LIN {X 0,Y 389.933,Z 569.817,A -85,B 0,C 180,E1 -11709.597,E2 -11709.597} C_VEL
LIN {X 0,Y 390.463,Z 562.006,A -85,B 0,C 180,E1 -11711.157,E2 -11711.157} C_VEL
LIN {X 0,Y 391.267,Z 552.298,A -85,B 0,C 180,E1 -11712.711,E2 -11712.711} C_VEL
LIN {X 0,Y 392.166,Z 541.336,A -85,B 0,C 180,E1 -11714.133,E2 -11714.133} C_VEL
LIN {X 0,Y 392.924,Z 530.148,A -85,B 0,C 180,E1 -11715.299,E2 -11715.299} C_VEL
LIN {X 0,Y 393.801,Z 517.877,A -85,B 0,C 180,E1 -11716.325,E2 -11716.325} C_VEL
LIN {X 0,Y 394.289,Z 508.273,A -85,B 0,C 180,E1 -11716.971,E2 -11716.971} C_VEL
LIN {X 0,Y 391.847,Z 495.073,A -85,B 0,C 180,E1 -11717.783,E2 -11717.783} C_VEL
LIN {X 0,Y 389.258,Z 482.057,A -85,B 0,C 180,E1 -11718.418,E2 -11718.418} C_VEL
LIN {X 0,Y 389.378,Z 477.403,A -85,B 0,C 180,E1 -11721.161,E2 -11721.161} C_VEL
LIN {X 0,Y 389.588,Z 471.826,A -85,B 0,C 180,E1 -11724.514,E2 -11724.514} C_VEL
LIN {X 0,Y 389.891,Z 466.202,A -85,B 0,C 180,E1 -11727.961,E2 -11727.961} C_VEL
LIN {X 0,Y 390.122,Z 460.557,A -85,B 0,C 180,E1 -11731.496,E2 -11731.496} C_VEL
LIN {X 0,Y 390.336,Z 456.52,A -85,B 0,C 180,E1 -11734.081,E2 -11734.081} C_VEL
LIN {X 0,Y 390.324,Z 452.898,A -85,B 0,C 180,E1 -11736.455,E2 -11736.455} C_VEL
LIN {X 0,Y 390.174,Z 450.511,A -85,B 0,C 180,E1 -11738.092,E2 -11738.092} C_VEL
LIN {X 0,Y 390.038,Z 450.527,A -85,B 0,C 180,E1 -11741.813,E2 -11741.813} C_VEL
LIN {X 0,Y 390.052,Z 450.528,A -85,B 0,C 180,E1 -11745.354,E2 -11745.354} C_VEL
LIN {X 0,Y 390.08,Z 450.612,A -85,B 0,C 180,E1 -11748.317,E2 -11748.317} C_VEL
LIN {X 0,Y 391.012,Z 456.192,A -85,B 0,C 180,E1 -11751.016,E2 -11751.016} C_VEL
LIN {X 0,Y 391.083,Z 460.373,A -85,B 0,C 180,E1 -11752.984,E2 -11752.984} C_VEL
LIN {X 0,Y 390.807,Z 467.118,A -85,B 0,C 180,E1 -11756.117,E2 -11756.117} C_VEL
LIN {X 0,Y 390.549,Z 473.709,A -85,B 0,C 180,E1 -11759.144,E2 -11759.144} C_VEL
LIN {X 0,Y 390.319,Z 480.242,A -85,B 0,C 180,E1 -11762.084,E2 -11762.084} C_VEL
LIN {X 0,Y 390.081,Z 486.796,A -85,B 0,C 180,E1 -11764.95,E2 -11764.95} C_VEL
LIN {X 0,Y 389.917,Z 492.999,A -85,B 0,C 180,E1 -11767.561,E2 -11767.561} C_VEL
LIN {X 0,Y 394.076,Z 508.813,A -85,B 0,C 180,E1 -11768.244,E2 -11768.244} C_VEL
LIN {X 0,Y 396.749,Z 522.313,A -85,B 0,C 180,E1 -11768.978,E2 -11768.978} C_VEL
LIN {X 0,Y 397.539,Z 527.293,A -85,B 0,C 180,E1 -11769.293,E2 -11769.293} C_VEL
LIN {X 0,Y 396.695,Z 539.579,A -85,B 0,C 180,E1 -11770.041,E2 -11770.041} C_VEL
LIN {X 0,Y 395.73,Z 551.412,A -85,B 0,C 180,E1 -11770.953,E2 -11770.953} C_VEL
LIN {X 0,Y 394.45,Z 563.522,A -85,B 0,C 180,E1 -11772.099,E2 -11772.099} C_VEL
LIN {X 0,Y 393.359,Z 574.511,A -85,B 0,C 180,E1 -11773.388,E2 -11773.388} C_VEL
LIN {X 0,Y 392.11,Z 585.305,A -85,B 0,C 180,E1 -11774.935,E2 -11774.935} C_VEL
LIN {X 0,Y 391.204,Z 594.223,A -85,B 0,C 180,E1 -11776.493,E2 -11776.493} C_VEL
LIN {X 0,Y 390.405,Z 601.649,A -85,B 0,C 180,E1 -11778.051,E2 -11778.051} C_VEL
LIN {X 0,Y 389.812,Z 607.841,A -85,B 0,C 180,E1 -11779.612,E2 -11779.612} C_VEL
LIN {X 0,Y 389.208,Z 614.385,A -85,B 0,C 180,E1 -11781.693,E2 -11781.693} C_VEL
LIN {X 0,Y 388.924,Z 619.291,A -85,B 0,C 180,E1 -11783.774,E2 -11783.774} C_VEL
LIN {X 0,Y 388.707,Z 622.712,A -85,B 0,C 180,E1 -11785.851,E2 -11785.851} C_VEL
LIN {X 0,Y 388.654,Z 624.749,A -85,B 0,C 180,E1 -11787.926,E2 -11787.926} C_VEL
LIN {X 0,Y 388.672,Z 625.452,A -85,B 0,C 180,E1 -11789.999,E2 -11789.999} C_VEL
LIN {X 0,Y 388.653,Z 624.824,A -85,B 0,C 180,E1 -11792.071,E2 -11792.071} C_VEL
LIN {X 0,Y 388.705,Z 622.851,A -85,B 0,C 180,E1 -11794.146,E2 -11794.146} C_VEL
LIN {X 0,Y 388.902,Z 619.492,A -85,B 0,C 180,E1 -11796.223,E2 -11796.223} C_VEL
LIN {X 0,Y 389.189,Z 614.648,A -85,B 0,C 180,E1 -11798.305,E2 -11798.305} C_VEL
LIN {X 0,Y 389.754,Z 608.177,A -85,B 0,C 180,E1 -11800.387,E2 -11800.387} C_VEL
LIN {X 0,Y 390.448,Z 601.498,A -85,B 0,C 180,E1 -11802.08,E2 -11802.08} C_VEL
LIN {X 0,Y 390.181,Z 598.35,A -85,B 0,C 180,E1 -11802.813,E2 -11802.813} C_VEL
LIN {X 0,Y 387.895,Z 592.988,A -85,B 0,C 180,E1 -11803.997,E2 -11803.997} C_VEL
LIN {X 0,Y 385.67,Z 587.106,A -85,B 0,C 180,E1 -11805.136,E2 -11805.136} C_VEL
LIN {X 0,Y 385.494,Z 583.143,A -85,B 0,C 180,E1 -11805.787,E2 -11805.787} C_VEL
LIN {X 0,Y 386.652,Z 573.256,A -85,B 0,C 180,E1 -11807.178,E2 -11807.178} C_VEL
LIN {X 0,Y 387.927,Z 561.979,A -85,B 0,C 180,E1 -11808.483,E2 -11808.483} C_VEL
LIN {X 0,Y 389.194,Z 549.516,A -85,B 0,C 180,E1 -11809.652,E2 -11809.652} C_VEL
LIN {X 0,Y 390.291,Z 536.229,A -85,B 0,C 180,E1 -11810.642,E2 -11810.642} C_VEL
LIN {X 0,Y 390.728,Z 527.81,A -85,B 0,C 180,E1 -11811.156,E2 -11811.156} C_VEL
LIN {X 0,Y 388.377,Z 514.529,A -85,B 0,C 180,E1 -11811.963,E2 -11811.963} C_VEL
LIN {X 0,Y 384.932,Z 500.27,A -85,B 0,C 180,E1 -11812.667,E2 -11812.667} C_VEL
LIN {X 0,Y 382.917,Z 493.014,A -85,B 0,C 180,E1 -11812.972,E2 -11812.972} C_VEL
LIN {X 0,Y 383.224,Z 484.334,A -85,B 0,C 180,E1 -11816.698,E2 -11816.698} C_VEL
LIN {X 0,Y 383.47,Z 477.73,A -85,B 0,C 180,E1 -11819.657,E2 -11819.657} C_VEL
LIN {X 0,Y 383.735,Z 469.811,A -85,B 0,C 180,E1 -11823.327,E2 -11823.327} C_VEL
LIN {X 0,Y 384.019,Z 463.336,A -85,B 0,C 180,E1 -11826.365,E2 -11826.365} C_VEL
LIN {X 0,Y 384.18,Z 458.893,A -85,B 0,C 180,E1 -11828.459,E2 -11828.459} C_VEL
LIN {X 0,Y 383.663,Z 454.572,A -85,B 0,C 180,E1 -11830.55,E2 -11830.55} C_VEL
LIN {X 0,Y 383.079,Z 451.397,A -85,B 0,C 180,E1 -11832.214,E2 -11832.214} C_VEL
LIN {X 0,Y 383.066,Z 451.397,A -85,B 0,C 180,E1 -11835.799,E2 -11835.799} C_VEL
LIN {X 0,Y 383.037,Z 451.399,A -85,B 0,C 180,E1 -11838.785,E2 -11838.785} C_VEL
LIN {X 0,Y 382.995,Z 451.401,A -85,B 0,C 180,E1 -11842.094,E2 -11842.094} C_VEL
LIN {X 0,Y 383.01,Z 451.396,A -85,B 0,C 180,E1 -11845.331,E2 -11845.331} C_VEL
LIN {X 0,Y 383.028,Z 451.401,A -85,B 0,C 180,E1 -11847.852,E2 -11847.852} C_VEL
LIN {X 0,Y 383.055,Z 451.396,A -85,B 0,C 180,E1 -11851.719,E2 -11851.719} C_VEL
LIN {X 0,Y 383.043,Z 451.397,A -85,B 0,C 180,E1 -11855.039,E2 -11855.039} C_VEL
LIN {X 0,Y 383.012,Z 451.39,A -85,B 0,C 180,E1 -11858.47,E2 -11858.47} C_VEL
LIN {X 0,Y 383.084,Z 451.392,A -85,B 0,C 180,E1 -11861.827,E2 -11861.827} C_VEL
LIN {X 0,Y 383.104,Z 451.387,A -85,B 0,C 180,E1 -11865.118,E2 -11865.118} C_VEL
LIN {X 0,Y 383.098,Z 451.385,A -85,B 0,C 180,E1 -11868.358,E2 -11868.358} C_VEL
LIN {X 0,Y 383.293,Z 451.361,A -85,B 0,C 180,E1 -11871.932,E2 -11871.932} C_VEL
LIN {X 0,Y 383.197,Z 451.373,A -85,B 0,C 180,E1 -11874.738,E2 -11874.738} C_VEL
LIN {X 0,Y 383.378,Z 451.352,A -85,B 0,C 180,E1 -11877.899,E2 -11877.899} C_VEL
LIN {X 0,Y 383.51,Z 451.338,A -85,B 0,C 180,E1 -11880,E2 -11880} C_VEL
LIN {X 0,Y 383.243,Z 451.353,A -85,B 0,C 180,E1 -11883.154,E2 -11883.154} C_VEL
LIN {X 0,Y 383.277,Z 451.367,A -85,B 0,C 180,E1 -11886.316,E2 -11886.316} C_VEL
LIN {X 0,Y 383.25,Z 451.367,A -85,B 0,C 180,E1 -11888.436,E2 -11888.436} C_VEL
LIN {X 0,Y 383.098,Z 451.375,A -85,B 0,C 180,E1 -11891.642,E2 -11891.642} C_VEL
LIN {X 0,Y 383.101,Z 451.39,A -85,B 0,C 180,E1 -11894.882,E2 -11894.882} C_VEL
LIN {X 0,Y 383.052,Z 451.38,A -85,B 0,C 180,E1 -11898.174,E2 -11898.174} C_VEL
LIN {X 0,Y 382.986,Z 451.404,A -85,B 0,C 180,E1 -11901.531,E2 -11901.531} C_VEL
LIN {X 0,Y 383.042,Z 451.396,A -85,B 0,C 180,E1 -11904.961,E2 -11904.961} C_VEL
LIN {X 0,Y 383.04,Z 451.395,A -85,B 0,C 180,E1 -11908.493,E2 -11908.493} C_VEL
LIN {X 0,Y 382.997,Z 451.406,A -85,B 0,C 180,E1 -11912.428,E2 -11912.428} C_VEL
LIN {X 0,Y 383.018,Z 451.4,A -85,B 0,C 180,E1 -11915.956,E2 -11915.956} C_VEL
LIN {X 0,Y 383.014,Z 451.402,A -85,B 0,C 180,E1 -11919.589,E2 -11919.589} C_VEL
LIN {X 0,Y 383.057,Z 451.398,A -85,B 0,C 180,E1 -11922.789,E2 -11922.789} C_VEL
LIN {X 0,Y 383,Z 451.403,A -85,B 0,C 180,E1 -11925.792,E2 -11925.792} C_VEL
LIN {X 0,Y 383.053,Z 451.529,A -85,B 0,C 180,E1 -11928.664,E2 -11928.664} C_VEL
LIN {X 0,Y 384.348,Z 458.285,A -85,B 0,C 180,E1 -11931.839,E2 -11931.839} C_VEL
LIN {X 0,Y 385.925,Z 466.782,A -85,B 0,C 180,E1 -11935.632,E2 -11935.632} C_VEL
LIN {X 0,Y 386.157,Z 469.798,A -85,B 0,C 180,E1 -11936.909,E2 -11936.909} C_VEL
LIN {X 0,Y 385.52,Z 475.759,A -85,B 0,C 180,E1 -11939.309,E2 -11939.309} C_VEL
LIN {X 0,Y 384.58,Z 484.683,A -85,B 0,C 180,E1 -11942.817,E2 -11942.817} C_VEL
LIN {X 0,Y 383.72,Z 493.805,A -85,B 0,C 180,E1 -11946.316,E2 -11946.316} C_VEL
LIN {X 0,Y 383.49,Z 496.446,A -85,B 0,C 180,E1 -11947.314,E2 -11947.314} C_VEL
LIN {X 0,Y 387.196,Z 513.156,A -85,B 0,C 180,E1 -11947.964,E2 -11947.964} C_VEL
LIN {X 0,Y 389.483,Z 526.876,A -85,B 0,C 180,E1 -11948.659,E2 -11948.659} C_VEL
LIN {X 0,Y 390.207,Z 534.647,A -85,B 0,C 180,E1 -11949.116,E2 -11949.116} C_VEL
LIN {X 0,Y 389.251,Z 547.706,A -85,B 0,C 180,E1 -11949.939,E2 -11949.939} C_VEL
LIN {X 0,Y 388.105,Z 560.544,A -85,B 0,C 180,E1 -11950.978,E2 -11950.978} C_VEL
LIN {X 0,Y 386.84,Z 572.176,A -85,B 0,C 180,E1 -11952.148,E2 -11952.148} C_VEL
LIN {X 0,Y 385.572,Z 583.784,A -85,B 0,C 180,E1 -11953.591,E2 -11953.591} C_VEL
LIN {X 0,Y 384.448,Z 594.141,A -85,B 0,C 180,E1 -11955.173,E2 -11955.173} C_VEL
LIN {X 0,Y 383.595,Z 602.664,A -85,B 0,C 180,E1 -11956.762,E2 -11956.762} C_VEL
LIN {X 0,Y 382.78,Z 610.781,A -85,B 0,C 180,E1 -11958.618,E2 -11958.618} C_VEL
LIN {X 0,Y 382.232,Z 617.299,A -85,B 0,C 180,E1 -11960.476,E2 -11960.476} C_VEL
LIN {X 0,Y 381.842,Z 623.064,A -85,B 0,C 180,E1 -11962.599,E2 -11962.599} C_VEL
LIN {X 0,Y 381.754,Z 625.601,A -85,B 0,C 180,E1 -11963.787,E2 -11963.787} C_VEL
LIN {X 0,Y 381.628,Z 628.789,A -85,B 0,C 180,E1 -11965.777,E2 -11965.777} C_VEL
LIN {X 0,Y 381.574,Z 630.823,A -85,B 0,C 180,E1 -11967.89,E2 -11967.89} C_VEL
LIN {X 0,Y 381.604,Z 631.498,A -85,B 0,C 180,E1 -11970.001,E2 -11970.001} C_VEL
LIN {X 0,Y 381.579,Z 630.815,A -85,B 0,C 180,E1 -11972.112,E2 -11972.112} C_VEL
LIN {X 0,Y 381.629,Z 628.772,A -85,B 0,C 180,E1 -11974.226,E2 -11974.226} C_VEL
LIN {X 0,Y 381.765,Z 625.324,A -85,B 0,C 180,E1 -11976.343,E2 -11976.343} C_VEL
LIN {X 0,Y 381.977,Z 620.365,A -85,B 0,C 180,E1 -11978.466,E2 -11978.466} C_VEL
LIN {X 0,Y 382.355,Z 615.547,A -85,B 0,C 180,E1 -11980.058,E2 -11980.058} C_VEL
LIN {X 0,Y 383.057,Z 608.575,A -85,B 0,C 180,E1 -11981.913,E2 -11981.913} C_VEL
LIN {X 0,Y 383.826,Z 599.915,A -85,B 0,C 180,E1 -11983.772,E2 -11983.772} C_VEL
LIN {X 0,Y 384.846,Z 590.834,A -85,B 0,C 180,E1 -11985.356,E2 -11985.356} C_VEL
LIN {X 0,Y 386.088,Z 579.795,A -85,B 0,C 180,E1 -11986.934,E2 -11986.934} C_VEL
LIN {X 0,Y 387.284,Z 568.483,A -85,B 0,C 180,E1 -11988.243,E2 -11988.243} C_VEL
LIN {X 0,Y 388.505,Z 556.144,A -85,B 0,C 180,E1 -11989.397,E2 -11989.397} C_VEL
LIN {X 0,Y 390.036,Z 542.056,A -85,B 0,C 180,E1 -11990.572,E2 -11990.572} C_VEL
LIN {X 0,Y 390.784,Z 533.606,A -85,B 0,C 180,E1 -11991.161,E2 -11991.161} C_VEL
LIN {X 0,Y 389.733,Z 521.037,A -85,B 0,C 180,E1 -11992.054,E2 -11992.054} C_VEL
LIN {X 0,Y 387.574,Z 509.699,A -85,B 0,C 180,E1 -11992.827,E2 -11992.827} C_VEL
LIN {X 0,Y 384.121,Z 497.15,A -85,B 0,C 180,E1 -11993.666,E2 -11993.666} C_VEL
LIN {X 0,Y 385.4,Z 488.006,A -85,B 0,C 180,E1 -11997.712,E2 -11997.712} C_VEL
LIN {X 0,Y 386.913,Z 480.633,A -85,B 0,C 180,E1 -12001.381,E2 -12001.381} C_VEL
LIN {X 0,Y 387.785,Z 476.845,A -85,B 0,C 180,E1 -12003.521,E2 -12003.521} C_VEL
LIN {X 0,Y 387.574,Z 474.066,A -85,B 0,C 180,E1 -12005.47,E2 -12005.47} C_VEL
LIN {X 0,Y 387.084,Z 470.987,A -85,B 0,C 180,E1 -12008.121,E2 -12008.121} C_VEL
LIN {X 0,Y 386.649,Z 468.636,A -85,B 0,C 180,E1 -12010.873,E2 -12010.873} C_VEL
LIN {X 0,Y 386.265,Z 467.097,A -85,B 0,C 180,E1 -12013.742,E2 -12013.742} C_VEL
LIN {X 0,Y 386.086,Z 466.459,A -85,B 0,C 180,E1 -12016.731,E2 -12016.731} C_VEL
LIN {X 0,Y 386.06,Z 466.782,A -85,B 0,C 180,E1 -12019.872,E2 -12019.872} C_VEL
LIN {X 0,Y 386.068,Z 467.443,A -85,B 0,C 180,E1 -12021.761,E2 -12021.761} C_VEL
LIN {X 0,Y 385.8,Z 468.927,A -85,B 0,C 180,E1 -12024.343,E2 -12024.343} C_VEL
LIN {X 0,Y 385.177,Z 471.124,A -85,B 0,C 180,E1 -12027.07,E2 -12027.07} C_VEL
LIN {X 0,Y 384.481,Z 474.436,A -85,B 0,C 180,E1 -12030.427,E2 -12030.427} C_VEL
LIN {X 0,Y 383.857,Z 478.463,A -85,B 0,C 180,E1 -12033.934,E2 -12033.934} C_VEL
LIN {X 0,Y 383.328,Z 482.836,A -85,B 0,C 180,E1 -12037.355,E2 -12037.355} C_VEL
LIN {X 0,Y 383.139,Z 485.087,A -85,B 0,C 180,E1 -12039.017,E2 -12039.017} C_VEL
LIN {X 0,Y 384.261,Z 488.308,A -85,B 0,C 180,E1 -12039.289,E2 -12039.289} C_VEL
LIN {X 0,Y 388.12,Z 500.175,A -85,B 0,C 180,E1 -12040.325,E2 -12040.325} C_VEL
LIN {X 0,Y 390.526,Z 510.382,A -85,B 0,C 180,E1 -12041.23,E2 -12041.23} C_VEL
LIN {X 0,Y 390.913,Z 514.795,A -85,B 0,C 180,E1 -12041.608,E2 -12041.608} C_VEL
LIN {X 0,Y 389.458,Z 527.72,A -85,B 0,C 180,E1 -12042.677,E2 -12042.677} C_VEL
LIN {X 0,Y 388.138,Z 539.334,A -85,B 0,C 180,E1 -12043.877,E2 -12043.877} C_VEL
LIN {X 0,Y 386.703,Z 550.212,A -85,B 0,C 180,E1 -12045.26,E2 -12045.26} C_VEL
LIN {X 0,Y 385.608,Z 558.633,A -85,B 0,C 180,E1 -12046.563,E2 -12046.563} C_VEL
LIN {X 0,Y 384.546,Z 567.011,A -85,B 0,C 180,E1 -12048.135,E2 -12048.135} C_VEL
LIN {X 0,Y 383.756,Z 573.896,A -85,B 0,C 180,E1 -12049.714,E2 -12049.714} C_VEL
LIN {X 0,Y 382.955,Z 580.232,A -85,B 0,C 180,E1 -12051.558,E2 -12051.558} C_VEL
LIN {X 0,Y 382.505,Z 584.537,A -85,B 0,C 180,E1 -12053.185,E2 -12053.185} C_VEL
LIN {X 0,Y 382.048,Z 587.618,A -85,B 0,C 180,E1 -12054.723,E2 -12054.723} C_VEL
LIN {X 0,Y 382.067,Z 589.17,A -85,B 0,C 180,E1 -12055.781,E2 -12055.781} C_VEL
LIN {X 0,Y 381.973,Z 590.339,A -85,B 0,C 180,E1 -12056.836,E2 -12056.836} C_VEL
LIN {X 0,Y 381.821,Z 591.097,A -85,B 0,C 180,E1 -12057.89,E2 -12057.89} C_VEL
LIN {X 0,Y 381.728,Z 591.416,A -85,B 0,C 180,E1 -12058.945,E2 -12058.945} C_VEL
LIN {X 0,Y 381.696,Z 591.335,A -85,B 0,C 180,E1 -12060,E2 -12060} C_VEL
LIN {X 0,Y 381.709,Z 590.856,A -85,B 0,C 180,E1 -12061.055,E2 -12061.055} C_VEL
LIN {X 0,Y 381.788,Z 589.968,A -85,B 0,C 180,E1 -12062.11,E2 -12062.11} C_VEL
LIN {X 0,Y 381.806,Z 588.633,A -85,B 0,C 180,E1 -12063.166,E2 -12063.166} C_VEL
LIN {X 0,Y 381.888,Z 585.855,A -85,B 0,C 180,E1 -12064.75,E2 -12064.75} C_VEL
LIN {X 0,Y 382.163,Z 580.884,A -85,B 0,C 180,E1 -12066.745,E2 -12066.745} C_VEL
LIN {X 0,Y 382.469,Z 575.217,A -85,B 0,C 180,E1 -12068.453,E2 -12068.453} C_VEL
LIN {X 0,Y 382.975,Z 568.566,A -85,B 0,C 180,E1 -12070.04,E2 -12070.04} C_VEL
LIN {X 0,Y 383.561,Z 560.345,A -85,B 0,C 180,E1 -12071.628,E2 -12071.628} C_VEL
LIN {X 0,Y 384.471,Z 550.229,A -85,B 0,C 180,E1 -12073.209,E2 -12073.209} C_VEL
LIN {X 0,Y 385.38,Z 539.776,A -85,B 0,C 180,E1 -12074.522,E2 -12074.522} C_VEL
LIN {X 0,Y 386.158,Z 528.392,A -85,B 0,C 180,E1 -12075.694,E2 -12075.694} C_VEL
LIN {X 0,Y 386.979,Z 517.197,A -85,B 0,C 180,E1 -12076.621,E2 -12076.621} C_VEL
LIN {X 0,Y 387.398,Z 509.517,A -85,B 0,C 180,E1 -12077.145,E2 -12077.145} C_VEL
LIN {X 0,Y 385.102,Z 496.919,A -85,B 0,C 180,E1 -12077.959,E2 -12077.959} C_VEL
LIN {X 0,Y 382.409,Z 483.603,A -85,B 0,C 180,E1 -12078.622,E2 -12078.622} C_VEL
LIN {X 0,Y 382.182,Z 482.184,A -85,B 0,C 180,E1 -12078.703,E2 -12078.703} C_VEL
LIN {X 0,Y 382.336,Z 477.404,A -85,B 0,C 180,E1 -12081.57,E2 -12081.57} C_VEL
LIN {X 0,Y 382.498,Z 473.675,A -85,B 0,C 180,E1 -12083.843,E2 -12083.843} C_VEL
LIN {X 0,Y 382.761,Z 468.037,A -85,B 0,C 180,E1 -12087.325,E2 -12087.325} C_VEL
LIN {X 0,Y 383.028,Z 462.359,A -85,B 0,C 180,E1 -12090.915,E2 -12090.915} C_VEL
LIN {X 0,Y 383.226,Z 458.546,A -85,B 0,C 180,E1 -12093.379,E2 -12093.379} C_VEL
LIN {X 0,Y 383.3,Z 454.249,A -85,B 0,C 180,E1 -12096.218,E2 -12096.218} C_VEL
LIN {X 0,Y 383.137,Z 451.387,A -85,B 0,C 180,E1 -12098.213,E2 -12098.213} C_VEL
LIN {X 0,Y 382.991,Z 451.405,A -85,B 0,C 180,E1 -12101.347,E2 -12101.347} C_VEL
LIN {X 0,Y 383.004,Z 451.402,A -85,B 0,C 180,E1 -12104.303,E2 -12104.303} C_VEL
LIN {X 0,Y 383.057,Z 451.53,A -85,B 0,C 180,E1 -12108.045,E2 -12108.045} C_VEL
LIN {X 0,Y 384.027,Z 457.32,A -85,B 0,C 180,E1 -12110.9,E2 -12110.9} C_VEL
LIN {X 0,Y 384.114,Z 461.422,A -85,B 0,C 180,E1 -12112.857,E2 -12112.857} C_VEL
LIN {X 0,Y 383.819,Z 468.277,A -85,B 0,C 180,E1 -12116.078,E2 -12116.078} C_VEL
LIN {X 0,Y 383.514,Z 475.58,A -85,B 0,C 180,E1 -12119.462,E2 -12119.462} C_VEL
LIN {X 0,Y 383.243,Z 482.773,A -85,B 0,C 180,E1 -12122.711,E2 -12122.711} C_VEL
LIN {X 0,Y 382.989,Z 490.775,A -85,B 0,C 180,E1 -12126.189,E2 -12126.189} C_VEL
LIN {X 0,Y 382.919,Z 493.02,A -85,B 0,C 180,E1 -12127.135,E2 -12127.135} C_VEL
LIN {X 0,Y 386.942,Z 508.181,A -85,B 0,C 180,E1 -12127.8,E2 -12127.8} C_VEL
LIN {X 0,Y 389.679,Z 521.173,A -85,B 0,C 180,E1 -12128.521,E2 -12128.521} C_VEL
LIN {X 0,Y 390.802,Z 529.215,A -85,B 0,C 180,E1 -12129.028,E2 -12129.028} C_VEL
LIN {X 0,Y 389.839,Z 541.992,A -85,B 0,C 180,E1 -12129.854,E2 -12129.854} C_VEL
LIN {X 0,Y 388.754,Z 554.364,A -85,B 0,C 180,E1 -12130.871,E2 -12130.871} C_VEL
LIN {X 0,Y 387.376,Z 565.903,A -85,B 0,C 180,E1 -12132.035,E2 -12132.035} C_VEL
LIN {X 0,Y 386.297,Z 576.479,A -85,B 0,C 180,E1 -12133.348,E2 -12133.348} C_VEL
LIN {X 0,Y 385.065,Z 586.956,A -85,B 0,C 180,E1 -12134.924,E2 -12134.924} C_VEL
LIN {X 0,Y 384.253,Z 594.277,A -85,B 0,C 180,E1 -12136.244,E2 -12136.244} C_VEL
LIN {X 0,Y 383.449,Z 601.704,A -85,B 0,C 180,E1 -12137.831,E2 -12137.831} C_VEL
LIN {X 0,Y 382.791,Z 607.896,A -85,B 0,C 180,E1 -12139.419,E2 -12139.419} C_VEL
LIN {X 0,Y 382.154,Z 614.441,A -85,B 0,C 180,E1 -12141.538,E2 -12141.538} C_VEL
LIN {X 0,Y 381.85,Z 619.347,A -85,B 0,C 180,E1 -12143.659,E2 -12143.659} C_VEL
LIN {X 0,Y 381.636,Z 622.768,A -85,B 0,C 180,E1 -12145.774,E2 -12145.774} C_VEL
LIN {X 0,Y 381.552,Z 624.805,A -85,B 0,C 180,E1 -12147.887,E2 -12147.887} C_VEL
LIN {X 0,Y 381.572,Z 625.508,A -85,B 0,C 180,E1 -12149.999,E2 -12149.999} C_VEL
LIN {X 0,Y 381.551,Z 624.879,A -85,B 0,C 180,E1 -12152.11,E2 -12152.11} C_VEL
LIN {X 0,Y 381.634,Z 622.906,A -85,B 0,C 180,E1 -12154.223,E2 -12154.223} C_VEL
LIN {X 0,Y 381.848,Z 619.546,A -85,B 0,C 180,E1 -12156.339,E2 -12156.339} C_VEL
LIN {X 0,Y 382.137,Z 614.701,A -85,B 0,C 180,E1 -12158.459,E2 -12158.459} C_VEL
LIN {X 0,Y 382.74,Z 608.229,A -85,B 0,C 180,E1 -12160.579,E2 -12160.579} C_VEL
LIN {X 0,Y 383.564,Z 601.013,A -85,B 0,C 180,E1 -12162.431,E2 -12162.431} C_VEL
LIN {X 0,Y 384.351,Z 593.036,A -85,B 0,C 180,E1 -12164.101,E2 -12164.101} C_VEL
LIN {X 0,Y 385.494,Z 583.143,A -85,B 0,C 180,E1 -12165.787,E2 -12165.787} C_VEL
LIN {X 0,Y 385.351,Z 579.067,A -85,B 0,C 180,E1 -12166.424,E2 -12166.424} C_VEL
LIN {X 0,Y 383.287,Z 572.294,A -85,B 0,C 180,E1 -12167.463,E2 -12167.463} C_VEL
LIN {X 0,Y 381.343,Z 565.192,A -85,B 0,C 180,E1 -12168.45,E2 -12168.45} C_VEL
LIN {X 0,Y 381.35,Z 560.456,A -85,B 0,C 180,E1 -12168.986,E2 -12168.986} C_VEL
LIN {X 0,Y 382.663,Z 548.011,A -85,B 0,C 180,E1 -12170.141,E2 -12170.141} C_VEL
LIN {X 0,Y 383.686,Z 535.454,A -85,B 0,C 180,E1 -12171.072,E2 -12171.072} C_VEL
LIN {X 0,Y 384.069,Z 529.092,A -85,B 0,C 180,E1 -12171.466,E2 -12171.466} C_VEL
LIN {X 0,Y 381.721,Z 515.792,A -85,B 0,C 180,E1 -12172.313,E2 -12172.313} C_VEL
LIN {X 0,Y 378.38,Z 501.769,A -85,B 0,C 180,E1 -12173.041,E2 -12173.041} C_VEL
LIN {X 0,Y 375.878,Z 492.976,A -85,B 0,C 180,E1 -12173.446,E2 -12173.446} C_VEL
LIN {X 0,Y 376.208,Z 485.605,A -85,B 0,C 180,E1 -12176.636,E2 -12176.636} C_VEL
LIN {X 0,Y 376.479,Z 477.591,A -85,B 0,C 180,E1 -12180.265,E2 -12180.265} C_VEL
LIN {X 0,Y 376.86,Z 469.586,A -85,B 0,C 180,E1 -12184.017,E2 -12184.017} C_VEL
LIN {X 0,Y 377.192,Z 461.355,A -85,B 0,C 180,E1 -12187.94,E2 -12187.94} C_VEL
LIN {X 0,Y 377.139,Z 458.516,A -85,B 0,C 180,E1 -12189.313,E2 -12189.313} C_VEL
LIN {X 0,Y 376.037,Z 452.273,A -85,B 0,C 180,E1 -12192.459,E2 -12192.459} C_VEL
LIN {X 0,Y 375.994,Z 452.277,A -85,B 0,C 180,E1 -12196.243,E2 -12196.243} C_VEL
LIN {X 0,Y 375.992,Z 452.273,A -85,B 0,C 180,E1 -12200.026,E2 -12200.026} C_VEL
LIN {X 0,Y 375.957,Z 452.281,A -85,B 0,C 180,E1 -12203.494,E2 -12203.494} C_VEL
LIN {X 0,Y 375.952,Z 452.275,A -85,B 0,C 180,E1 -12205.888,E2 -12205.888} C_VEL
LIN {X 0,Y 375.966,Z 452.273,A -85,B 0,C 180,E1 -12209.687,E2 -12209.687} C_VEL
LIN {X 0,Y 375.993,Z 452.272,A -85,B 0,C 180,E1 -12212.141,E2 -12212.141} C_VEL
LIN {X 0,Y 375.997,Z 452.271,A -85,B 0,C 180,E1 -12214.538,E2 -12214.538} C_VEL
LIN {X 0,Y 375.975,Z 452.265,A -85,B 0,C 180,E1 -12218.046,E2 -12218.046} C_VEL
LIN {X 0,Y 376.022,Z 452.27,A -85,B 0,C 180,E1 -12221.474,E2 -12221.474} C_VEL
LIN {X 0,Y 376.052,Z 452.264,A -85,B 0,C 180,E1 -12224.832,E2 -12224.832} C_VEL
LIN {X 0,Y 376.049,Z 452.263,A -85,B 0,C 180,E1 -12228.136,E2 -12228.136} C_VEL
LIN {X 0,Y 376.247,Z 452.238,A -85,B 0,C 180,E1 -12231.876,E2 -12231.876} C_VEL
LIN {X 0,Y 376.169,Z 452.249,A -85,B 0,C 180,E1 -12234.64,E2 -12234.64} C_VEL
LIN {X 0,Y 376.344,Z 452.228,A -85,B 0,C 180,E1 -12237.859,E2 -12237.859} C_VEL
LIN {X 0,Y 376.48,Z 452.214,A -85,B 0,C 180,E1 -12240,E2 -12240} C_VEL
LIN {X 0,Y 376.181,Z 452.232,A -85,B 0,C 180,E1 -12243.213,E2 -12243.213} C_VEL
LIN {X 0,Y 376.236,Z 452.245,A -85,B 0,C 180,E1 -12246.435,E2 -12246.435} C_VEL
LIN {X 0,Y 376.195,Z 452.244,A -85,B 0,C 180,E1 -12248.595,E2 -12248.595} C_VEL
LIN {X 0,Y 376.05,Z 452.256,A -85,B 0,C 180,E1 -12251.863,E2 -12251.863} C_VEL
LIN {X 0,Y 376.049,Z 452.265,A -85,B 0,C 180,E1 -12255.168,E2 -12255.168} C_VEL
LIN {X 0,Y 375.998,Z 452.262,A -85,B 0,C 180,E1 -12258.527,E2 -12258.527} C_VEL
LIN {X 0,Y 375.954,Z 452.278,A -85,B 0,C 180,E1 -12261.955,E2 -12261.955} C_VEL
LIN {X 0,Y 375.996,Z 452.273,A -85,B 0,C 180,E1 -12265.462,E2 -12265.462} C_VEL
LIN {X 0,Y 375.967,Z 452.28,A -85,B 0,C 180,E1 -12269.079,E2 -12269.079} C_VEL
LIN {X 0,Y 375.945,Z 452.281,A -85,B 0,C 180,E1 -12272.829,E2 -12272.829} C_VEL
LIN {X 0,Y 375.949,Z 452.282,A -85,B 0,C 180,E1 -12275.416,E2 -12275.416} C_VEL
LIN {X 0,Y 375.969,Z 452.277,A -85,B 0,C 180,E1 -12278.272,E2 -12278.272} C_VEL
LIN {X 0,Y 375.982,Z 452.275,A -85,B 0,C 180,E1 -12281.611,E2 -12281.611} C_VEL
LIN {X 0,Y 375.961,Z 452.279,A -85,B 0,C 180,E1 -12285.263,E2 -12285.263} C_VEL
LIN {X 0,Y 376.006,Z 452.321,A -85,B 0,C 180,E1 -12288.292,E2 -12288.292} C_VEL
LIN {X 0,Y 377.269,Z 458.962,A -85,B 0,C 180,E1 -12291.481,E2 -12291.481} C_VEL
LIN {X 0,Y 378.663,Z 466.369,A -85,B 0,C 180,E1 -12294.877,E2 -12294.877} C_VEL
LIN {X 0,Y 379.179,Z 470.11,A -85,B 0,C 180,E1 -12296.519,E2 -12296.519} C_VEL
LIN {X 0,Y 378.477,Z 476.853,A -85,B 0,C 180,E1 -12299.295,E2 -12299.295} C_VEL
LIN {X 0,Y 377.519,Z 485.767,A -85,B 0,C 180,E1 -12302.867,E2 -12302.867} C_VEL
LIN {X 0,Y 376.537,Z 495.84,A -85,B 0,C 180,E1 -12306.805,E2 -12306.805} C_VEL
LIN {X 0,Y 376.516,Z 495.994,A -85,B 0,C 180,E1 -12306.864,E2 -12306.864} C_VEL
LIN {X 0,Y 380.27,Z 512.854,A -85,B 0,C 180,E1 -12307.53,E2 -12307.53} C_VEL
LIN {X 0,Y 382.547,Z 526.044,A -85,B 0,C 180,E1 -12308.214,E2 -12308.214} C_VEL
LIN {X 0,Y 383.481,Z 535.862,A -85,B 0,C 180,E1 -12308.809,E2 -12308.809} C_VEL
LIN {X 0,Y 382.426,Z 549.332,A -85,B 0,C 180,E1 -12309.697,E2 -12309.697} C_VEL
LIN {X 0,Y 381.211,Z 561.927,A -85,B 0,C 180,E1 -12310.761,E2 -12310.761} C_VEL
LIN {X 0,Y 379.945,Z 573.304,A -85,B 0,C 180,E1 -12311.953,E2 -12311.953} C_VEL
LIN {X 0,Y 378.723,Z 583.738,A -85,B 0,C 180,E1 -12313.285,E2 -12313.285} C_VEL
LIN {X 0,Y 377.544,Z 594.093,A -85,B 0,C 180,E1 -12314.895,E2 -12314.895} C_VEL
LIN {X 0,Y 376.613,Z 602.614,A -85,B 0,C 180,E1 -12316.512,E2 -12316.512} C_VEL
LIN {X 0,Y 375.963,Z 609.679,A -85,B 0,C 180,E1 -12318.135,E2 -12318.135} C_VEL
LIN {X 0,Y 375.328,Z 615.525,A -85,B 0,C 180,E1 -12319.755,E2 -12319.755} C_VEL
LIN {X 0,Y 374.824,Z 621.755,A -85,B 0,C 180,E1 -12321.917,E2 -12321.917} C_VEL
LIN {X 0,Y 374.681,Z 625.788,A -85,B 0,C 180,E1 -12323.792,E2 -12323.792} C_VEL
LIN {X 0,Y 374.554,Z 628.734,A -85,B 0,C 180,E1 -12325.697,E2 -12325.697} C_VEL
LIN {X 0,Y 374.471,Z 630.768,A -85,B 0,C 180,E1 -12327.85,E2 -12327.85} C_VEL
LIN {X 0,Y 374.505,Z 631.442,A -85,B 0,C 180,E1 -12330.001,E2 -12330.001} C_VEL
LIN {X 0,Y 374.476,Z 630.759,A -85,B 0,C 180,E1 -12332.152,E2 -12332.152} C_VEL
LIN {X 0,Y 374.555,Z 628.716,A -85,B 0,C 180,E1 -12334.306,E2 -12334.306} C_VEL
LIN {X 0,Y 374.678,Z 625.268,A -85,B 0,C 180,E1 -12336.463,E2 -12336.463} C_VEL
LIN {X 0,Y 374.937,Z 620.309,A -85,B 0,C 180,E1 -12338.626,E2 -12338.626} C_VEL
LIN {X 0,Y 375.325,Z 615.492,A -85,B 0,C 180,E1 -12340.248,E2 -12340.248} C_VEL
LIN {X 0,Y 376.071,Z 608.52,A -85,B 0,C 180,E1 -12342.138,E2 -12342.138} C_VEL
LIN {X 0,Y 376.878,Z 599.861,A -85,B 0,C 180,E1 -12344.031,E2 -12344.031} C_VEL
LIN {X 0,Y 377.949,Z 590.782,A -85,B 0,C 180,E1 -12345.643,E2 -12345.643} C_VEL
LIN {X 0,Y 379.272,Z 579.745,A -85,B 0,C 180,E1 -12347.248,E2 -12347.248} C_VEL
LIN {X 0,Y 380.541,Z 568.436,A -85,B 0,C 180,E1 -12348.578,E2 -12348.578} C_VEL
LIN {X 0,Y 382.625,Z 550.606,A -85,B 0,C 180,E1 -12350.32,E2 -12350.32} C_VEL
LIN {X 0,Y 384.035,Z 538.034,A -85,B 0,C 180,E1 -12351.33,E2 -12351.33} C_VEL
LIN {X 0,Y 384.284,Z 533.8,A -85,B 0,C 180,E1 -12351.637,E2 -12351.637} C_VEL
LIN {X 0,Y 383.237,Z 521.314,A -85,B 0,C 180,E1 -12352.571,E2 -12352.571} C_VEL
LIN {X 0,Y 380.871,Z 509.274,A -85,B 0,C 180,E1 -12353.447,E2 -12353.447} C_VEL
LIN {X 0,Y 377.305,Z 496.933,A -85,B 0,C 180,E1 -12354.347,E2 -12354.347} C_VEL
LIN {X 0,Y 378.649,Z 488.468,A -85,B 0,C 180,E1 -12358.25,E2 -12358.25} C_VEL
LIN {X 0,Y 380.166,Z 481.722,A -85,B 0,C 180,E1 -12361.746,E2 -12361.746} C_VEL
LIN {X 0,Y 380.903,Z 478.169,A -85,B 0,C 180,E1 -12363.871,E2 -12363.871} C_VEL
LIN {X 0,Y 380.583,Z 475.047,A -85,B 0,C 180,E1 -12366.224,E2 -12366.224} C_VEL
LIN {X 0,Y 380.106,Z 472.099,A -85,B 0,C 180,E1 -12369.053,E2 -12369.053} C_VEL
LIN {X 0,Y 379.744,Z 470.073,A -85,B 0,C 180,E1 -12371.78,E2 -12371.78} C_VEL
LIN {X 0,Y 379.35,Z 468.688,A -85,B 0,C 180,E1 -12375.251,E2 -12375.251} C_VEL
LIN {X 0,Y 379.235,Z 468.476,A -85,B 0,C 180,E1 -12378.152,E2 -12378.152} C_VEL
LIN {X 0,Y 379.218,Z 469.106,A -85,B 0,C 180,E1 -12381.114,E2 -12381.114} C_VEL
LIN {X 0,Y 379.043,Z 470.289,A -85,B 0,C 180,E1 -12383.607,E2 -12383.607} C_VEL
LIN {X 0,Y 378.492,Z 472.083,A -85,B 0,C 180,E1 -12386.148,E2 -12386.148} C_VEL
LIN {X 0,Y 377.911,Z 474.426,A -85,B 0,C 180,E1 -12388.812,E2 -12388.812} C_VEL
LIN {X 0,Y 377.174,Z 477.99,A -85,B 0,C 180,E1 -12392.236,E2 -12392.236} C_VEL
LIN {X 0,Y 376.555,Z 482.153,A -85,B 0,C 180,E1 -12395.757,E2 -12395.757} C_VEL
LIN {X 0,Y 376.216,Z 485.454,A -85,B 0,C 180,E1 -12398.313,E2 -12398.313} C_VEL
LIN {X 0,Y 377.397,Z 488.77,A -85,B 0,C 180,E1 -12398.612,E2 -12398.612} C_VEL
LIN {X 0,Y 381.522,Z 500.709,A -85,B 0,C 180,E1 -12399.742,E2 -12399.742} C_VEL
LIN {X 0,Y 384.021,Z 511.523,A -85,B 0,C 180,E1 -12400.767,E2 -12400.767} C_VEL
LIN {X 0,Y 384.529,Z 514.759,A -85,B 0,C 180,E1 -12401.076,E2 -12401.076} C_VEL
LIN {X 0,Y 383.223,Z 527.091,A -85,B 0,C 180,E1 -12402.111,E2 -12402.111} C_VEL
LIN {X 0,Y 381.645,Z 539.707,A -85,B 0,C 180,E1 -12403.432,E2 -12403.432} C_VEL
LIN {X 0,Y 380.287,Z 549.725,A -85,B 0,C 180,E1 -12404.731,E2 -12404.731} C_VEL
LIN {X 0,Y 378.804,Z 559.814,A -85,B 0,C 180,E1 -12406.317,E2 -12406.317} C_VEL
LIN {X 0,Y 377.697,Z 568.062,A -85,B 0,C 180,E1 -12407.917,E2 -12407.917} C_VEL
LIN {X 0,Y 376.829,Z 574.75,A -85,B 0,C 180,E1 -12409.523,E2 -12409.523} C_VEL
LIN {X 0,Y 375.99,Z 580.958,A -85,B 0,C 180,E1 -12411.4,E2 -12411.4} C_VEL
LIN {X 0,Y 375.572,Z 584.292,A -85,B 0,C 180,E1 -12412.654,E2 -12412.654} C_VEL
LIN {X 0,Y 375.003,Z 588.2,A -85,B 0,C 180,E1 -12414.623,E2 -12414.623} C_VEL
LIN {X 0,Y 375.005,Z 589.711,A -85,B 0,C 180,E1 -12415.701,E2 -12415.701} C_VEL
LIN {X 0,Y 374.921,Z 590.832,A -85,B 0,C 180,E1 -12416.776,E2 -12416.776} C_VEL
LIN {X 0,Y 374.762,Z 591.521,A -85,B 0,C 180,E1 -12417.851,E2 -12417.851} C_VEL
LIN {X 0,Y 374.627,Z 591.684,A -85,B 0,C 180,E1 -12420,E2 -12420} C_VEL
LIN {X 0,Y 374.643,Z 591.17,A -85,B 0,C 180,E1 -12421.075,E2 -12421.075} C_VEL
LIN {X 0,Y 374.707,Z 590.221,A -85,B 0,C 180,E1 -12422.15,E2 -12422.15} C_VEL
LIN {X 0,Y 374.711,Z 588.846,A -85,B 0,C 180,E1 -12423.226,E2 -12423.226} C_VEL
LIN {X 0,Y 374.829,Z 585.993,A -85,B 0,C 180,E1 -12424.84,E2 -12424.84} C_VEL
LIN {X 0,Y 375.092,Z 581.269,A -85,B 0,C 180,E1 -12426.753,E2 -12426.753} C_VEL
LIN {X 0,Y 375.41,Z 575.155,A -85,B 0,C 180,E1 -12428.614,E2 -12428.614} C_VEL
LIN {X 0,Y 375.952,Z 568.39,A -85,B 0,C 180,E1 -12430.23,E2 -12430.23} C_VEL
LIN {X 0,Y 376.576,Z 560.066,A -85,B 0,C 180,E1 -12431.847,E2 -12431.847} C_VEL
LIN {X 0,Y 377.35,Z 551.668,A -85,B 0,C 180,E1 -12433.188,E2 -12433.188} C_VEL
LIN {X 0,Y 378.239,Z 541.612,A -85,B 0,C 180,E1 -12434.52,E2 -12434.52} C_VEL
LIN {X 0,Y 379.071,Z 530.362,A -85,B 0,C 180,E1 -12435.732,E2 -12435.732} C_VEL
LIN {X 0,Y 379.987,Z 518.08,A -85,B 0,C 180,E1 -12436.798,E2 -12436.798} C_VEL
LIN {X 0,Y 380.432,Z 510.231,A -85,B 0,C 180,E1 -12437.354,E2 -12437.354} C_VEL
LIN {X 0,Y 377.992,Z 496.888,A -85,B 0,C 180,E1 -12438.232,E2 -12438.232} C_VEL
LIN {X 0,Y 375.246,Z 483.362,A -85,B 0,C 180,E1 -12438.913,E2 -12438.913} C_VEL
LIN {X 0,Y 375.119,Z 482.312,A -85,B 0,C 180,E1 -12438.998,E2 -12438.998} C_VEL
LIN {X 0,Y 375.313,Z 477.395,A -85,B 0,C 180,E1 -12441.994,E2 -12441.994} C_VEL
LIN {X 0,Y 375.542,Z 471.755,A -85,B 0,C 180,E1 -12445.495,E2 -12445.495} C_VEL
LIN {X 0,Y 375.846,Z 466.077,A -85,B 0,C 180,E1 -12449.09,E2 -12449.09} C_VEL
LIN {X 0,Y 376.153,Z 460.341,A -85,B 0,C 180,E1 -12452.809,E2 -12452.809} C_VEL
LIN {X 0,Y 376.248,Z 456.476,A -85,B 0,C 180,E1 -12455.384,E2 -12455.384} C_VEL
LIN {X 0,Y 376.104,Z 452.264,A -85,B 0,C 180,E1 -12458.294,E2 -12458.294} C_VEL
LIN {X 0,Y 375.938,Z 452.282,A -85,B 0,C 180,E1 -12462.3,E2 -12462.3} C_VEL
LIN {X 0,Y 375.96,Z 452.284,A -85,B 0,C 180,E1 -12465.264,E2 -12465.264} C_VEL
LIN {X 0,Y 376.024,Z 452.352,A -85,B 0,C 180,E1 -12467.711,E2 -12467.711} C_VEL
LIN {X 0,Y 377.02,Z 458.232,A -85,B 0,C 180,E1 -12470.668,E2 -12470.668} C_VEL
LIN {X 0,Y 377.154,Z 462.473,A -85,B 0,C 180,E1 -12472.722,E2 -12472.722} C_VEL
LIN {X 0,Y 376.846,Z 469.325,A -85,B 0,C 180,E1 -12475.978,E2 -12475.978} C_VEL
LIN {X 0,Y 376.482,Z 477.349,A -85,B 0,C 180,E1 -12479.732,E2 -12479.732} C_VEL
LIN {X 0,Y 376.186,Z 485.357,A -85,B 0,C 180,E1 -12483.359,E2 -12483.359} C_VEL
LIN {X 0,Y 375.929,Z 493.024,A -85,B 0,C 180,E1 -12486.685,E2 -12486.685} C_VEL
LIN {X 0,Y 380.041,Z 508.281,A -85,B 0,C 180,E1 -12487.378,E2 -12487.378} C_VEL
LIN {X 0,Y 382.773,Z 520.99,A -85,B 0,C 180,E1 -12488.103,E2 -12488.103} C_VEL
LIN {X 0,Y 384.074,Z 529.372,A -85,B 0,C 180,E1 -12488.651,E2 -12488.651} C_VEL
LIN {X 0,Y 383.147,Z 542.418,A -85,B 0,C 180,E1 -12489.518,E2 -12489.518} C_VEL
LIN {X 0,Y 382.037,Z 554.41,A -85,B 0,C 180,E1 -12490.522,E2 -12490.522} C_VEL
LIN {X 0,Y 380.495,Z 567.1,A -85,B 0,C 180,E1 -12491.837,E2 -12491.837} C_VEL
LIN {X 0,Y 379.234,Z 578.444,A -85,B 0,C 180,E1 -12493.306,E2 -12493.306} C_VEL
LIN {X 0,Y 377.995,Z 588.604,A -85,B 0,C 180,E1 -12494.911,E2 -12494.911} C_VEL
LIN {X 0,Y 377.215,Z 595.663,A -85,B 0,C 180,E1 -12496.257,E2 -12496.257} C_VEL
LIN {X 0,Y 376.326,Z 602.858,A -85,B 0,C 180,E1 -12497.871,E2 -12497.871} C_VEL
LIN {X 0,Y 375.586,Z 609.735,A -85,B 0,C 180,E1 -12499.759,E2 -12499.759} C_VEL
LIN {X 0,Y 375,Z 615.9,A -85,B 0,C 180,E1 -12501.918,E2 -12501.918} C_VEL
LIN {X 0,Y 374.768,Z 619.665,A -85,B 0,C 180,E1 -12503.673,E2 -12503.673} C_VEL
LIN {X 0,Y 374.566,Z 622.824,A -85,B 0,C 180,E1 -12505.694,E2 -12505.694} C_VEL
LIN {X 0,Y 374.45,Z 624.861,A -85,B 0,C 180,E1 -12507.847,E2 -12507.847} C_VEL
LIN {X 0,Y 374.473,Z 625.564,A -85,B 0,C 180,E1 -12509.999,E2 -12509.999} C_VEL
LIN {X 0,Y 374.449,Z 624.935,A -85,B 0,C 180,E1 -12512.15,E2 -12512.15} C_VEL
LIN {X 0,Y 374.564,Z 622.961,A -85,B 0,C 180,E1 -12514.303,E2 -12514.303} C_VEL
LIN {X 0,Y 374.78,Z 619.6,A -85,B 0,C 180,E1 -12516.459,E2 -12516.459} C_VEL
LIN {X 0,Y 375.098,Z 614.755,A -85,B 0,C 180,E1 -12518.619,E2 -12518.619} C_VEL
LIN {X 0,Y 375.709,Z 608.281,A -85,B 0,C 180,E1 -12520.78,E2 -12520.78} C_VEL
LIN {X 0,Y 376.598,Z 601.064,A -85,B 0,C 180,E1 -12522.665,E2 -12522.665} C_VEL
LIN {X 0,Y 377.539,Z 592.175,A -85,B 0,C 180,E1 -12524.534,E2 -12524.534} C_VEL
LIN {X 0,Y 378.703,Z 582.669,A -85,B 0,C 180,E1 -12526.161,E2 -12526.161} C_VEL
LIN {X 0,Y 379.986,Z 572.252,A -85,B 0,C 180,E1 -12527.628,E2 -12527.628} C_VEL
LIN {X 0,Y 381.35,Z 560.456,A -85,B 0,C 180,E1 -12528.986,E2 -12528.986} C_VEL
LIN {X 0,Y 381.348,Z 555.635,A -85,B 0,C 180,E1 -12529.502,E2 -12529.502} C_VEL
LIN {X 0,Y 379.375,Z 547.759,A -85,B 0,C 180,E1 -12530.369,E2 -12530.369} C_VEL
LIN {X 0,Y 377.324,Z 539.552,A -85,B 0,C 180,E1 -12531.158,E2 -12531.158} C_VEL
LIN {X 0,Y 377.181,Z 534.217,A -85,B 0,C 180,E1 -12531.541,E2 -12531.541} C_VEL
LIN {X 0,Y 377.231,Z 529.11,A -85,B 0,C 180,E1 -12531.875,E2 -12531.875} C_VEL
LIN {X 0,Y 374.758,Z 515.304,A -85,B 0,C 180,E1 -12532.772,E2 -12532.772} C_VEL
LIN {X 0,Y 371.308,Z 501.37,A -85,B 0,C 180,E1 -12533.515,E2 -12533.515} C_VEL
LIN {X 0,Y 368.906,Z 493.005,A -85,B 0,C 180,E1 -12533.903,E2 -12533.903} C_VEL
LIN {X 0,Y 369.229,Z 485.54,A -85,B 0,C 180,E1 -12537.18,E2 -12537.18} C_VEL
LIN {X 0,Y 369.481,Z 478.795,A -85,B 0,C 180,E1 -12540.267,E2 -12540.267} C_VEL
LIN {X 0,Y 369.882,Z 470.694,A -85,B 0,C 180,E1 -12544.09,E2 -12544.09} C_VEL
LIN {X 0,Y 370.18,Z 463.87,A -85,B 0,C 180,E1 -12547.409,E2 -12547.409} C_VEL
LIN {X 0,Y 370.134,Z 459.588,A -85,B 0,C 180,E1 -12549.498,E2 -12549.498} C_VEL
LIN {X 0,Y 368.997,Z 453.15,A -85,B 0,C 180,E1 -12552.792,E2 -12552.792} C_VEL
LIN {X 0,Y 368.968,Z 453.152,A -85,B 0,C 180,E1 -12556.368,E2 -12556.368} C_VEL
LIN {X 0,Y 368.945,Z 453.154,A -85,B 0,C 180,E1 -12559.634,E2 -12559.634} C_VEL
LIN {X 0,Y 368.895,Z 453.158,A -85,B 0,C 180,E1 -12563.143,E2 -12563.143} C_VEL
LIN {X 0,Y 368.891,Z 453.159,A -85,B 0,C 180,E1 -12566.461,E2 -12566.461} C_VEL
LIN {X 0,Y 368.919,Z 453.158,A -85,B 0,C 180,E1 -12570.31,E2 -12570.31} C_VEL
LIN {X 0,Y 368.972,Z 453.142,A -85,B 0,C 180,E1 -12573.534,E2 -12573.534} C_VEL
LIN {X 0,Y 368.969,Z 453.15,A -85,B 0,C 180,E1 -12576.422,E2 -12576.422} C_VEL
LIN {X 0,Y 368.946,Z 453.15,A -85,B 0,C 180,E1 -12579.947,E2 -12579.947} C_VEL
LIN {X 0,Y 368.969,Z 453.149,A -85,B 0,C 180,E1 -12583.398,E2 -12583.398} C_VEL
LIN {X 0,Y 369.049,Z 453.14,A -85,B 0,C 180,E1 -12586.79,E2 -12586.79} C_VEL
LIN {X 0,Y 369.062,Z 453.138,A -85,B 0,C 180,E1 -12590.131,E2 -12590.131} C_VEL
LIN {X 0,Y 369.178,Z 453.122,A -85,B 0,C 180,E1 -12592.342,E2 -12592.342} C_VEL
LIN {X 0,Y 369.142,Z 453.125,A -85,B 0,C 180,E1 -12594.537,E2 -12594.537} C_VEL
LIN {X 0,Y 369.309,Z 453.105,A -85,B 0,C 180,E1 -12597.819,E2 -12597.819} C_VEL
LIN {X 0,Y 369.449,Z 453.09,A -85,B 0,C 180,E1 -12600,E2 -12600} C_VEL
LIN {X 0,Y 369.309,Z 453.1,A -85,B 0,C 180,E1 -12602.181,E2 -12602.181} C_VEL
LIN {X 0,Y 369.198,Z 453.123,A -85,B 0,C 180,E1 -12606.558,E2 -12606.558} C_VEL
LIN {X 0,Y 369.128,Z 453.124,A -85,B 0,C 180,E1 -12608.761,E2 -12608.761} C_VEL
LIN {X 0,Y 369.004,Z 453.137,A -85,B 0,C 180,E1 -12612.093,E2 -12612.093} C_VEL
LIN {X 0,Y 368.988,Z 453.142,A -85,B 0,C 180,E1 -12615.465,E2 -12615.465} C_VEL
LIN {X 0,Y 368.948,Z 453.145,A -85,B 0,C 180,E1 -12618.895,E2 -12618.895} C_VEL
LIN {X 0,Y 368.923,Z 453.154,A -85,B 0,C 180,E1 -12622.396,E2 -12622.396} C_VEL
LIN {X 0,Y 368.99,Z 453.147,A -85,B 0,C 180,E1 -12625.981,E2 -12625.981} C_VEL
LIN {X 0,Y 368.958,Z 453.151,A -85,B 0,C 180,E1 -12628.814,E2 -12628.814} C_VEL
LIN {X 0,Y 368.894,Z 453.161,A -85,B 0,C 180,E1 -12632.238,E2 -12632.238} C_VEL
LIN {X 0,Y 368.92,Z 453.156,A -85,B 0,C 180,E1 -12635.003,E2 -12635.003} C_VEL
LIN {X 0,Y 368.905,Z 453.157,A -85,B 0,C 180,E1 -12638.642,E2 -12638.642} C_VEL
LIN {X 0,Y 368.934,Z 453.153,A -85,B 0,C 180,E1 -12642.021,E2 -12642.021} C_VEL
LIN {X 0,Y 368.916,Z 453.157,A -85,B 0,C 180,E1 -12645.184,E2 -12645.184} C_VEL
LIN {X 0,Y 368.949,Z 453.23,A -85,B 0,C 180,E1 -12647.979,E2 -12647.979} C_VEL
LIN {X 0,Y 370.221,Z 459.828,A -85,B 0,C 180,E1 -12651.214,E2 -12651.214} C_VEL
LIN {X 0,Y 371.728,Z 467.832,A -85,B 0,C 180,E1 -12654.957,E2 -12654.957} C_VEL
LIN {X 0,Y 372.189,Z 470.564,A -85,B 0,C 180,E1 -12656.186,E2 -12656.186} C_VEL
LIN {X 0,Y 371.599,Z 476.726,A -85,B 0,C 180,E1 -12658.785,E2 -12658.785} C_VEL
LIN {X 0,Y 370.43,Z 486.82,A -85,B 0,C 180,E1 -12662.915,E2 -12662.915} C_VEL
LIN {X 0,Y 369.558,Z 495.464,A -85,B 0,C 180,E1 -12666.37,E2 -12666.37} C_VEL
LIN {X 0,Y 373.573,Z 513.45,A -85,B 0,C 180,E1 -12667.123,E2 -12667.123} C_VEL
LIN {X 0,Y 375.762,Z 526.184,A -85,B 0,C 180,E1 -12667.807,E2 -12667.807} C_VEL
LIN {X 0,Y 376.817,Z 536.515,A -85,B 0,C 180,E1 -12668.459,E2 -12668.459} C_VEL
LIN {X 0,Y 375.667,Z 550.285,A -85,B 0,C 180,E1 -12669.395,E2 -12669.395} C_VEL
LIN {X 0,Y 374.512,Z 561.89,A -85,B 0,C 180,E1 -12670.402,E2 -12670.402} C_VEL
LIN {X 0,Y 373.047,Z 574.431,A -85,B 0,C 180,E1 -12671.749,E2 -12671.749} C_VEL
LIN {X 0,Y 371.693,Z 585.575,A -85,B 0,C 180,E1 -12673.243,E2 -12673.243} C_VEL
LIN {X 0,Y 370.422,Z 595.693,A -85,B 0,C 180,E1 -12674.908,E2 -12674.908} C_VEL
LIN {X 0,Y 369.547,Z 603.915,A -85,B 0,C 180,E1 -12676.555,E2 -12676.555} C_VEL
LIN {X 0,Y 368.671,Z 611.683,A -85,B 0,C 180,E1 -12678.455,E2 -12678.455} C_VEL
LIN {X 0,Y 368.139,Z 617.192,A -85,B 0,C 180,E1 -12680.108,E2 -12680.108} C_VEL
LIN {X 0,Y 367.68,Z 622.955,A -85,B 0,C 180,E1 -12682.312,E2 -12682.312} C_VEL
LIN {X 0,Y 367.597,Z 625.996,A -85,B 0,C 180,E1 -12683.813,E2 -12683.813} C_VEL
LIN {X 0,Y 367.46,Z 628.679,A -85,B 0,C 180,E1 -12685.614,E2 -12685.614} C_VEL
LIN {X 0,Y 367.371,Z 630.712,A -85,B 0,C 180,E1 -12687.809,E2 -12687.809} C_VEL
LIN {X 0,Y 367.406,Z 631.386,A -85,B 0,C 180,E1 -12690.001,E2 -12690.001} C_VEL
LIN {X 0,Y 367.376,Z 630.703,A -85,B 0,C 180,E1 -12692.194,E2 -12692.194} C_VEL
LIN {X 0,Y 367.461,Z 628.661,A -85,B 0,C 180,E1 -12694.389,E2 -12694.389} C_VEL
LIN {X 0,Y 367.588,Z 625.212,A -85,B 0,C 180,E1 -12696.589,E2 -12696.589} C_VEL
LIN {X 0,Y 367.873,Z 620.253,A -85,B 0,C 180,E1 -12698.793,E2 -12698.793} C_VEL
LIN {X 0,Y 368.305,Z 615.436,A -85,B 0,C 180,E1 -12700.446,E2 -12700.446} C_VEL
LIN {X 0,Y 369.065,Z 608.465,A -85,B 0,C 180,E1 -12702.372,E2 -12702.372} C_VEL
LIN {X 0,Y 369.935,Z 599.671,A -85,B 0,C 180,E1 -12704.328,E2 -12704.328} C_VEL
LIN {X 0,Y 371.098,Z 590.73,A -85,B 0,C 180,E1 -12705.94,E2 -12705.94} C_VEL
LIN {X 0,Y 372.484,Z 579.695,A -85,B 0,C 180,E1 -12707.572,E2 -12707.572} C_VEL
LIN {X 0,Y 373.807,Z 568.393,A -85,B 0,C 180,E1 -12708.926,E2 -12708.926} C_VEL
LIN {X 0,Y 375.558,Z 555.192,A -85,B 0,C 180,E1 -12710.359,E2 -12710.359} C_VEL
LIN {X 0,Y 377.353,Z 541.301,A -85,B 0,C 180,E1 -12711.583,E2 -12711.583} C_VEL
LIN {X 0,Y 377.892,Z 535.261,A -85,B 0,C 180,E1 -12712.044,E2 -12712.044} C_VEL
LIN {X 0,Y 377.081,Z 523.757,A -85,B 0,C 180,E1 -12712.961,E2 -12712.961} C_VEL
LIN {X 0,Y 375.053,Z 512.539,A -85,B 0,C 180,E1 -12713.836,E2 -12713.836} C_VEL
LIN {X 0,Y 371.44,Z 499.91,A -85,B 0,C 180,E1 -12714.837,E2 -12714.837} C_VEL
LIN {X 0,Y 370.548,Z 496.622,A -85,B 0,C 180,E1 -12715.122,E2 -12715.122} C_VEL
LIN {X 0,Y 371.937,Z 488.966,A -85,B 0,C 180,E1 -12718.807,E2 -12718.807} C_VEL
LIN {X 0,Y 373.428,Z 482.845,A -85,B 0,C 180,E1 -12722.123,E2 -12722.123} C_VEL
LIN {X 0,Y 373.82,Z 481.313,A -85,B 0,C 180,E1 -12723.041,E2 -12723.041} C_VEL
LIN {X 0,Y 373.983,Z 479.397,A -85,B 0,C 180,E1 -12724.318,E2 -12724.318} C_VEL
LIN {X 0,Y 373.603,Z 476.09,A -85,B 0,C 180,E1 -12727.012,E2 -12727.012} C_VEL
LIN {X 0,Y 373.182,Z 473.466,A -85,B 0,C 180,E1 -12729.816,E2 -12729.816} C_VEL
LIN {X 0,Y 372.779,Z 471.611,A -85,B 0,C 180,E1 -12732.744,E2 -12732.744} C_VEL
LIN {X 0,Y 372.517,Z 470.612,A -85,B 0,C 180,E1 -12735.802,E2 -12735.802} C_VEL
LIN {X 0,Y 372.398,Z 470.559,A -85,B 0,C 180,E1 -12739.017,E2 -12739.017} C_VEL
LIN {X 0,Y 372.345,Z 471.17,A -85,B 0,C 180,E1 -12741.474,E2 -12741.474} C_VEL
LIN {X 0,Y 372.089,Z 472.475,A -85,B 0,C 180,E1 -12744.16,E2 -12744.16} C_VEL
LIN {X 0,Y 371.475,Z 474.31,A -85,B 0,C 180,E1 -12746.725,E2 -12746.725} C_VEL
LIN {X 0,Y 370.897,Z 476.502,A -85,B 0,C 180,E1 -12749.229,E2 -12749.229} C_VEL
LIN {X 0,Y 370.055,Z 480.614,A -85,B 0,C 180,E1 -12753.205,E2 -12753.205} C_VEL
LIN {X 0,Y 369.395,Z 485.162,A -85,B 0,C 180,E1 -12757.044,E2 -12757.044} C_VEL
LIN {X 0,Y 369.361,Z 486.011,A -85,B 0,C 180,E1 -12757.559,E2 -12757.559} C_VEL
LIN {X 0,Y 370.615,Z 489.266,A -85,B 0,C 180,E1 -12757.891,E2 -12757.891} C_VEL
LIN {X 0,Y 374.585,Z 500.233,A -85,B 0,C 180,E1 -12759.012,E2 -12759.012} C_VEL
LIN {X 0,Y 377.394,Z 511.523,A -85,B 0,C 180,E1 -12760.148,E2 -12760.148} C_VEL
LIN {X 0,Y 378.204,Z 517.486,A -85,B 0,C 180,E1 -12760.741,E2 -12760.741} C_VEL
LIN {X 0,Y 376.629,Z 529.552,A -85,B 0,C 180,E1 -12761.815,E2 -12761.815} C_VEL
LIN {X 0,Y 375.03,Z 541.447,A -85,B 0,C 180,E1 -12763.131,E2 -12763.131} C_VEL
LIN {X 0,Y 373.268,Z 553.04,A -85,B 0,C 180,E1 -12764.717,E2 -12764.717} C_VEL
LIN {X 0,Y 372.018,Z 561.069,A -85,B 0,C 180,E1 -12766.062,E2 -12766.062} C_VEL
LIN {X 0,Y 370.845,Z 569.072,A -85,B 0,C 180,E1 -12767.69,E2 -12767.69} C_VEL
LIN {X 0,Y 369.759,Z 576.625,A -85,B 0,C 180,E1 -12769.597,E2 -12769.597} C_VEL
LIN {X 0,Y 369.03,Z 581.749,A -85,B 0,C 180,E1 -12771.237,E2 -12771.237} C_VEL
LIN {X 0,Y 368.57,Z 585.056,A -85,B 0,C 180,E1 -12772.553,E2 -12772.553} C_VEL
LIN {X 0,Y 367.961,Z 588.781,A -85,B 0,C 180,E1 -12774.52,E2 -12774.52} C_VEL
LIN {X 0,Y 367.946,Z 590.256,A -85,B 0,C 180,E1 -12775.618,E2 -12775.618} C_VEL
LIN {X 0,Y 367.87,Z 591.319,A -85,B 0,C 180,E1 -12776.714,E2 -12776.714} C_VEL
LIN {X 0,Y 367.704,Z 591.954,A -85,B 0,C 180,E1 -12777.809,E2 -12777.809} C_VEL
LIN {X 0,Y 367.596,Z 592.193,A -85,B 0,C 180,E1 -12778.905,E2 -12778.905} C_VEL
LIN {X 0,Y 367.56,Z 592.035,A -85,B 0,C 180,E1 -12780,E2 -12780} C_VEL
LIN {X 0,Y 367.579,Z 591.469,A -85,B 0,C 180,E1 -12781.096,E2 -12781.096} C_VEL
LIN {X 0,Y 367.612,Z 590.46,A -85,B 0,C 180,E1 -12782.191,E2 -12782.191} C_VEL
LIN {X 0,Y 367.617,Z 589.047,A -85,B 0,C 180,E1 -12783.288,E2 -12783.288} C_VEL
LIN {X 0,Y 367.77,Z 586.122,A -85,B 0,C 180,E1 -12784.933,E2 -12784.933} C_VEL
LIN {X 0,Y 368.005,Z 581.047,A -85,B 0,C 180,E1 -12786.977,E2 -12786.977} C_VEL
LIN {X 0,Y 368.376,Z 575.077,A -85,B 0,C 180,E1 -12788.779,E2 -12788.779} C_VEL
LIN {X 0,Y 368.939,Z 568.213,A -85,B 0,C 180,E1 -12790.426,E2 -12790.426} C_VEL
LIN {X 0,Y 369.604,Z 559.777,A -85,B 0,C 180,E1 -12792.073,E2 -12792.073} C_VEL
LIN {X 0,Y 370.416,Z 551.266,A -85,B 0,C 180,E1 -12793.44,E2 -12793.44} C_VEL
LIN {X 0,Y 371.292,Z 541.474,A -85,B 0,C 180,E1 -12794.743,E2 -12794.743} C_VEL
LIN {X 0,Y 372.172,Z 529.598,A -85,B 0,C 180,E1 -12796.032,E2 -12796.032} C_VEL
LIN {X 0,Y 373.153,Z 517.07,A -85,B 0,C 180,E1 -12797.115,E2 -12797.115} C_VEL
LIN {X 0,Y 373.323,Z 510.366,A -85,B 0,C 180,E1 -12797.601,E2 -12797.601} C_VEL
LIN {X 0,Y 370.897,Z 496.967,A -85,B 0,C 180,E1 -12798.504,E2 -12798.504} C_VEL
LIN {X 0,Y 368.061,Z 482.514,A -85,B 0,C 180,E1 -12799.268,E2 -12799.268} C_VEL
LIN {X 0,Y 368.261,Z 477.372,A -85,B 0,C 180,E1 -12802.438,E2 -12802.438} C_VEL
LIN {X 0,Y 368.586,Z 471.187,A -85,B 0,C 180,E1 -12806.339,E2 -12806.339} C_VEL
LIN {X 0,Y 368.83,Z 465.989,A -85,B 0,C 180,E1 -12809.698,E2 -12809.698} C_VEL
LIN {X 0,Y 369.121,Z 460.831,A -85,B 0,C 180,E1 -12813.095,E2 -12813.095} C_VEL
LIN {X 0,Y 369.194,Z 456.311,A -85,B 0,C 180,E1 -12816.166,E2 -12816.166} C_VEL
LIN {X 0,Y 369.047,Z 453.143,A -85,B 0,C 180,E1 -12818.379,E2 -12818.379} C_VEL
LIN {X 0,Y 368.888,Z 453.161,A -85,B 0,C 180,E1 -12822.009,E2 -12822.009} C_VEL
LIN {X 0,Y 368.933,Z 453.159,A -85,B 0,C 180,E1 -12825.183,E2 -12825.183} C_VEL
LIN {X 0,Y 368.987,Z 453.196,A -85,B 0,C 180,E1 -12827.377,E2 -12827.377} C_VEL
LIN {X 0,Y 370.008,Z 459.3,A -85,B 0,C 180,E1 -12830.483,E2 -12830.483} C_VEL
LIN {X 0,Y 370.183,Z 463.557,A -85,B 0,C 180,E1 -12832.588,E2 -12832.588} C_VEL
LIN {X 0,Y 369.871,Z 470.457,A -85,B 0,C 180,E1 -12835.906,E2 -12835.906} C_VEL
LIN {X 0,Y 369.539,Z 477.212,A -85,B 0,C 180,E1 -12839.102,E2 -12839.102} C_VEL
LIN {X 0,Y 369.27,Z 483.936,A -85,B 0,C 180,E1 -12842.205,E2 -12842.205} C_VEL
LIN {X 0,Y 368.943,Z 491.928,A -85,B 0,C 180,E1 -12845.74,E2 -12845.74} C_VEL
LIN {X 0,Y 368.923,Z 493.022,A -85,B 0,C 180,E1 -12846.212,E2 -12846.212} C_VEL
LIN {X 0,Y 373.224,Z 508.596,A -85,B 0,C 180,E1 -12846.952,E2 -12846.952} C_VEL
LIN {X 0,Y 376.149,Z 522.568,A -85,B 0,C 180,E1 -12847.777,E2 -12847.777} C_VEL
LIN {X 0,Y 377.32,Z 529.541,A -85,B 0,C 180,E1 -12848.258,E2 -12848.258} C_VEL
LIN {X 0,Y 376.502,Z 542.266,A -85,B 0,C 180,E1 -12849.123,E2 -12849.123} C_VEL
LIN {X 0,Y 375.335,Z 554.456,A -85,B 0,C 180,E1 -12850.159,E2 -12850.159} C_VEL
LIN {X 0,Y 373.712,Z 567.149,A -85,B 0,C 180,E1 -12851.496,E2 -12851.496} C_VEL
LIN {X 0,Y 372.411,Z 578.495,A -85,B 0,C 180,E1 -12852.99,E2 -12852.99} C_VEL
LIN {X 0,Y 371.097,Z 588.657,A -85,B 0,C 180,E1 -12854.624,E2 -12854.624} C_VEL
LIN {X 0,Y 370.161,Z 597.044,A -85,B 0,C 180,E1 -12856.27,E2 -12856.27} C_VEL
LIN {X 0,Y 369.043,Z 605.053,A -85,B 0,C 180,E1 -12858.186,E2 -12858.186} C_VEL
LIN {X 0,Y 368.38,Z 611.496,A -85,B 0,C 180,E1 -12860.112,E2 -12860.112} C_VEL
LIN {X 0,Y 367.844,Z 617.2,A -85,B 0,C 180,E1 -12862.313,E2 -12862.313} C_VEL
LIN {X 0,Y 367.691,Z 619.968,A -85,B 0,C 180,E1 -12863.681,E2 -12863.681} C_VEL
LIN {X 0,Y 367.476,Z 622.88,A -85,B 0,C 180,E1 -12865.611,E2 -12865.611} C_VEL
LIN {X 0,Y 367.352,Z 624.917,A -85,B 0,C 180,E1 -12867.806,E2 -12867.806} C_VEL
LIN {X 0,Y 367.373,Z 625.619,A -85,B 0,C 180,E1 -12869.999,E2 -12869.999} C_VEL
LIN {X 0,Y 367.35,Z 624.99,A -85,B 0,C 180,E1 -12872.191,E2 -12872.191} C_VEL
LIN {X 0,Y 367.474,Z 623.016,A -85,B 0,C 180,E1 -12874.386,E2 -12874.386} C_VEL
LIN {X 0,Y 367.694,Z 619.655,A -85,B 0,C 180,E1 -12876.584,E2 -12876.584} C_VEL
LIN {X 0,Y 368.048,Z 614.808,A -85,B 0,C 180,E1 -12878.786,E2 -12878.786} C_VEL
LIN {X 0,Y 368.686,Z 608.334,A -85,B 0,C 180,E1 -12880.988,E2 -12880.988} C_VEL
LIN {X 0,Y 369.636,Z 601.115,A -85,B 0,C 180,E1 -12882.908,E2 -12882.908} C_VEL
LIN {X 0,Y 370.583,Z 592.739,A -85,B 0,C 180,E1 -12884.714,E2 -12884.714} C_VEL
LIN {X 0,Y 371.868,Z 582.715,A -85,B 0,C 180,E1 -12886.467,E2 -12886.467} C_VEL
LIN {X 0,Y 373.189,Z 572.295,A -85,B 0,C 180,E1 -12887.96,E2 -12887.96} C_VEL
LIN {X 0,Y 374.599,Z 560.795,A -85,B 0,C 180,E1 -12889.308,E2 -12889.308} C_VEL
LIN {X 0,Y 375.992,Z 548.043,A -85,B 0,C 180,E1 -12890.515,E2 -12890.515} C_VEL
LIN {X 0,Y 377.17,Z 534.33,A -85,B 0,C 180,E1 -12891.534,E2 -12891.534} C_VEL
LIN {X 0,Y 377.181,Z 534.217,A -85,B 0,C 180,E1 -12891.541,E2 -12891.541} C_VEL
LIN {X 0,Y 377.069,Z 530.662,A -85,B 0,C 180,E1 -12891.782,E2 -12891.782} C_VEL
LIN {X 0,Y 376.129,Z 527.296,A -85,B 0,C 180,E1 -12892.051,E2 -12892.051} C_VEL
LIN {X 0,Y 372.85,Z 521.056,A -85,B 0,C 180,E1 -12892.618,E2 -12892.618} C_VEL
LIN {X 0,Y 368.088,Z 513.192,A -85,B 0,C 180,E1 -12893.31,E2 -12893.31} C_VEL
LIN {X 0,Y 366.115,Z 507.88,A -85,B 0,C 180,E1 -12893.65,E2 -12893.65} C_VEL
LIN {X 0,Y 361.914,Z 492.989,A -85,B 0,C 180,E1 -12894.401,E2 -12894.401} C_VEL
LIN {X 0,Y 362.278,Z 485.466,A -85,B 0,C 180,E1 -12897.746,E2 -12897.746} C_VEL
LIN {X 0,Y 362.596,Z 477.457,A -85,B 0,C 180,E1 -12901.479,E2 -12901.479} C_VEL
LIN {X 0,Y 362.965,Z 470.471,A -85,B 0,C 180,E1 -12904.832,E2 -12904.832} C_VEL
LIN {X 0,Y 363.264,Z 463.536,A -85,B 0,C 180,E1 -12908.248,E2 -12908.248} C_VEL
LIN {X 0,Y 362.954,Z 459.443,A -85,B 0,C 180,E1 -12910.298,E2 -12910.298} C_VEL
LIN {X 0,Y 361.924,Z 454.03,A -85,B 0,C 180,E1 -12913.194,E2 -12913.194} C_VEL
LIN {X 0,Y 361.923,Z 454.03,A -85,B 0,C 180,E1 -12915.927,E2 -12915.927} C_VEL
LIN {X 0,Y 361.898,Z 454.035,A -85,B 0,C 180,E1 -12919.23,E2 -12919.23} C_VEL
LIN {X 0,Y 361.861,Z 454.033,A -85,B 0,C 180,E1 -12922.981,E2 -12922.981} C_VEL
LIN {X 0,Y 361.854,Z 454.037,A -85,B 0,C 180,E1 -12926.629,E2 -12926.629} C_VEL
LIN {X 0,Y 361.87,Z 454.028,A -85,B 0,C 180,E1 -12929.671,E2 -12929.671} C_VEL
LIN {X 0,Y 361.945,Z 454.017,A -85,B 0,C 180,E1 -12933.474,E2 -12933.474} C_VEL
LIN {X 0,Y 361.895,Z 454.022,A -85,B 0,C 180,E1 -12937.145,E2 -12937.145} C_VEL
LIN {X 0,Y 361.923,Z 454.028,A -85,B 0,C 180,E1 -12940.724,E2 -12940.724} C_VEL
LIN {X 0,Y 361.939,Z 454.024,A -85,B 0,C 180,E1 -12944.226,E2 -12944.226} C_VEL
LIN {X 0,Y 361.99,Z 454.018,A -85,B 0,C 180,E1 -12946.527,E2 -12946.527} C_VEL
LIN {X 0,Y 362.026,Z 454.014,A -85,B 0,C 180,E1 -12949.938,E2 -12949.938} C_VEL
LIN {X 0,Y 362.141,Z 453.997,A -85,B 0,C 180,E1 -12952.192,E2 -12952.192} C_VEL
LIN {X 0,Y 362.115,Z 454,A -85,B 0,C 180,E1 -12954.431,E2 -12954.431} C_VEL
LIN {X 0,Y 362.273,Z 453.981,A -85,B 0,C 180,E1 -12957.776,E2 -12957.776} C_VEL
LIN {X 0,Y 362.419,Z 453.965,A -85,B 0,C 180,E1 -12960,E2 -12960} C_VEL
LIN {X 0,Y 362.273,Z 453.976,A -85,B 0,C 180,E1 -12962.224,E2 -12962.224} C_VEL
LIN {X 0,Y 362.161,Z 453.999,A -85,B 0,C 180,E1 -12966.686,E2 -12966.686} C_VEL
LIN {X 0,Y 362.065,Z 454.003,A -85,B 0,C 180,E1 -12968.933,E2 -12968.933} C_VEL
LIN {X 0,Y 361.957,Z 454.017,A -85,B 0,C 180,E1 -12972.332,E2 -12972.332} C_VEL
LIN {X 0,Y 361.952,Z 454.024,A -85,B 0,C 180,E1 -12974.621,E2 -12974.621} C_VEL
LIN {X 0,Y 361.945,Z 454.008,A -85,B 0,C 180,E1 -12978.1,E2 -12978.1} C_VEL
LIN {X 0,Y 361.882,Z 454.033,A -85,B 0,C 180,E1 -12981.654,E2 -12981.654} C_VEL
LIN {X 0,Y 361.918,Z 454.027,A -85,B 0,C 180,E1 -12985.291,E2 -12985.291} C_VEL
LIN {X 0,Y 361.913,Z 454.026,A -85,B 0,C 180,E1 -12987.779,E2 -12987.779} C_VEL
LIN {X 0,Y 361.838,Z 454.036,A -85,B 0,C 180,E1 -12991.286,E2 -12991.286} C_VEL
LIN {X 0,Y 361.846,Z 454.038,A -85,B 0,C 180,E1 -12994.281,E2 -12994.281} C_VEL
LIN {X 0,Y 361.864,Z 454.034,A -85,B 0,C 180,E1 -12997.226,E2 -12997.226} C_VEL
LIN {X 0,Y 361.897,Z 454.032,A -85,B 0,C 180,E1 -13000.769,E2 -13000.769} C_VEL
LIN {X 0,Y 361.896,Z 454.033,A -85,B 0,C 180,E1 -13004.356,E2 -13004.356} C_VEL
LIN {X 0,Y 361.912,Z 454.132,A -85,B 0,C 180,E1 -13007.653,E2 -13007.653} C_VEL
LIN {X 0,Y 363.275,Z 461.319,A -85,B 0,C 180,E1 -13011.256,E2 -13011.256} C_VEL
LIN {X 0,Y 364.618,Z 468.503,A -85,B 0,C 180,E1 -13014.675,E2 -13014.675} C_VEL
LIN {X 0,Y 365.148,Z 471.533,A -85,B 0,C 180,E1 -13016.073,E2 -13016.073} C_VEL
LIN {X 0,Y 364.851,Z 475.846,A -85,B 0,C 180,E1 -13017.947,E2 -13017.947} C_VEL
LIN {X 0,Y 363.675,Z 484.881,A -85,B 0,C 180,E1 -13021.743,E2 -13021.743} C_VEL
LIN {X 0,Y 362.663,Z 494.315,A -85,B 0,C 180,E1 -13025.617,E2 -13025.617} C_VEL
LIN {X 0,Y 362.607,Z 494.985,A -85,B 0,C 180,E1 -13025.888,E2 -13025.888} C_VEL
LIN {X 0,Y 366.608,Z 512.559,A -85,B 0,C 180,E1 -13026.632,E2 -13026.632} C_VEL
LIN {X 0,Y 369.021,Z 526.339,A -85,B 0,C 180,E1 -13027.387,E2 -13027.387} C_VEL
LIN {X 0,Y 370.188,Z 536.495,A -85,B 0,C 180,E1 -13028.054,E2 -13028.054} C_VEL
LIN {X 0,Y 369.049,Z 549.919,A -85,B 0,C 180,E1 -13028.981,E2 -13028.981} C_VEL
LIN {X 0,Y 367.832,Z 561.853,A -85,B 0,C 180,E1 -13030.032,E2 -13030.032} C_VEL
LIN {X 0,Y 366.294,Z 574.389,A -85,B 0,C 180,E1 -13031.4,E2 -13031.4} C_VEL
LIN {X 0,Y 364.865,Z 585.529,A -85,B 0,C 180,E1 -13032.919,E2 -13032.919} C_VEL
LIN {X 0,Y 363.55,Z 595.496,A -85,B 0,C 180,E1 -13034.587,E2 -13034.587} C_VEL
LIN {X 0,Y 362.56,Z 603.876,A -85,B 0,C 180,E1 -13036.293,E2 -13036.293} C_VEL
LIN {X 0,Y 361.696,Z 611.631,A -85,B 0,C 180,E1 -13038.229,E2 -13038.229} C_VEL
LIN {X 0,Y 361.116,Z 617.139,A -85,B 0,C 180,E1 -13039.914,E2 -13039.914} C_VEL
LIN {X 0,Y 360.629,Z 622.901,A -85,B 0,C 180,E1 -13042.161,E2 -13042.161} C_VEL
LIN {X 0,Y 360.412,Z 627.084,A -85,B 0,C 180,E1 -13044.406,E2 -13044.406} C_VEL
LIN {X 0,Y 360.302,Z 629.812,A -85,B 0,C 180,E1 -13046.647,E2 -13046.647} C_VEL
LIN {X 0,Y 360.313,Z 631.163,A -85,B 0,C 180,E1 -13048.884,E2 -13048.884} C_VEL
LIN {X 0,Y 360.315,Z 631.159,A -85,B 0,C 180,E1 -13051.119,E2 -13051.119} C_VEL
LIN {X 0,Y 360.302,Z 629.797,A -85,B 0,C 180,E1 -13053.356,E2 -13053.356} C_VEL
LIN {X 0,Y 360.412,Z 627.061,A -85,B 0,C 180,E1 -13055.597,E2 -13055.597} C_VEL
LIN {X 0,Y 360.632,Z 622.874,A -85,B 0,C 180,E1 -13057.842,E2 -13057.842} C_VEL
LIN {X 0,Y 361.116,Z 617.105,A -85,B 0,C 180,E1 -13060.089,E2 -13060.089} C_VEL
LIN {X 0,Y 361.842,Z 610.58,A -85,B 0,C 180,E1 -13062.053,E2 -13062.053} C_VEL
LIN {X 0,Y 362.698,Z 602.662,A -85,B 0,C 180,E1 -13063.972,E2 -13063.972} C_VEL
LIN {X 0,Y 363.785,Z 593.923,A -85,B 0,C 180,E1 -13065.693,E2 -13065.693} C_VEL
LIN {X 0,Y 365.153,Z 583.557,A -85,B 0,C 180,E1 -13067.358,E2 -13067.358} C_VEL
LIN {X 0,Y 367.774,Z 564.565,A -85,B 0,C 180,E1 -13069.829,E2 -13069.829} C_VEL
LIN {X 0,Y 369.68,Z 551.842,A -85,B 0,C 180,E1 -13071.176,E2 -13071.176} C_VEL
LIN {X 0,Y 371.499,Z 538.105,A -85,B 0,C 180,E1 -13072.35,E2 -13072.35} C_VEL
LIN {X 0,Y 371,Z 526.678,A -85,B 0,C 180,E1 -13073.316,E2 -13073.316} C_VEL
LIN {X 0,Y 369.314,Z 516.033,A -85,B 0,C 180,E1 -13074.212,E2 -13074.212} C_VEL
LIN {X 0,Y 366.183,Z 503.885,A -85,B 0,C 180,E1 -13075.245,E2 -13075.245} C_VEL
LIN {X 0,Y 363.797,Z 496.463,A -85,B 0,C 180,E1 -13075.896,E2 -13075.896} C_VEL
LIN {X 0,Y 365.22,Z 489.534,A -85,B 0,C 180,E1 -13079.388,E2 -13079.388} C_VEL
LIN {X 0,Y 366.677,Z 484.016,A -85,B 0,C 180,E1 -13082.506,E2 -13082.506} C_VEL
LIN {X 0,Y 367.092,Z 480.922,A -85,B 0,C 180,E1 -13084.59,E2 -13084.59} C_VEL
LIN {X 0,Y 366.876,Z 478.68,A -85,B 0,C 180,E1 -13086.432,E2 -13086.432} C_VEL
LIN {X 0,Y 366.437,Z 475.919,A -85,B 0,C 180,E1 -13089.267,E2 -13089.267} C_VEL
LIN {X 0,Y 366.025,Z 473.918,A -85,B 0,C 180,E1 -13092.225,E2 -13092.225} C_VEL
LIN {X 0,Y 365.721,Z 472.756,A -85,B 0,C 180,E1 -13095.32,E2 -13095.32} C_VEL
LIN {X 0,Y 365.601,Z 472.495,A -85,B 0,C 180,E1 -13098.566,E2 -13098.566} C_VEL
LIN {X 0,Y 365.583,Z 472.838,A -85,B 0,C 180,E1 -13100.625,E2 -13100.625} C_VEL
LIN {X 0,Y 365.333,Z 473.917,A -85,B 0,C 180,E1 -13103.391,E2 -13103.391} C_VEL
LIN {X 0,Y 364.767,Z 475.569,A -85,B 0,C 180,E1 -13106.031,E2 -13106.031} C_VEL
LIN {X 0,Y 364.141,Z 477.622,A -85,B 0,C 180,E1 -13108.594,E2 -13108.594} C_VEL
LIN {X 0,Y 363.266,Z 481.234,A -85,B 0,C 180,E1 -13112.334,E2 -13112.334} C_VEL
LIN {X 0,Y 362.594,Z 485.302,A -85,B 0,C 180,E1 -13115.981,E2 -13115.981} C_VEL
LIN {X 0,Y 362.484,Z 486.244,A -85,B 0,C 180,E1 -13116.713,E2 -13116.713} C_VEL
LIN {X 0,Y 363.725,Z 489.564,A -85,B 0,C 180,E1 -13117.064,E2 -13117.064} C_VEL
LIN {X 0,Y 367.837,Z 500.297,A -85,B 0,C 180,E1 -13118.283,E2 -13118.283} C_VEL
LIN {X 0,Y 370.672,Z 511.004,A -85,B 0,C 180,E1 -13119.428,E2 -13119.428} C_VEL
LIN {X 0,Y 371.926,Z 518.677,A -85,B 0,C 180,E1 -13120.259,E2 -13120.259} C_VEL
LIN {X 0,Y 370.161,Z 531.635,A -85,B 0,C 180,E1 -13121.457,E2 -13121.457} C_VEL
LIN {X 0,Y 368.423,Z 543.294,A -85,B 0,C 180,E1 -13122.82,E2 -13122.82} C_VEL
LIN {X 0,Y 366.59,Z 554.496,A -85,B 0,C 180,E1 -13124.431,E2 -13124.431} C_VEL
LIN {X 0,Y 365.247,Z 562.362,A -85,B 0,C 180,E1 -13125.799,E2 -13125.799} C_VEL
LIN {X 0,Y 364.019,Z 570.177,A -85,B 0,C 180,E1 -13127.455,E2 -13127.455} C_VEL
LIN {X 0,Y 362.842,Z 577.538,A -85,B 0,C 180,E1 -13129.397,E2 -13129.397} C_VEL
LIN {X 0,Y 362.075,Z 582.559,A -85,B 0,C 180,E1 -13131.067,E2 -13131.067} C_VEL
LIN {X 0,Y 361.534,Z 585.952,A -85,B 0,C 180,E1 -13132.491,E2 -13132.491} C_VEL
LIN {X 0,Y 360.922,Z 589.4,A -85,B 0,C 180,E1 -13134.413,E2 -13134.413} C_VEL
LIN {X 0,Y 360.875,Z 590.816,A -85,B 0,C 180,E1 -13135.532,E2 -13135.532} C_VEL
LIN {X 0,Y 360.802,Z 591.794,A -85,B 0,C 180,E1 -13136.65,E2 -13136.65} C_VEL
LIN {X 0,Y 360.649,Z 592.384,A -85,B 0,C 180,E1 -13137.766,E2 -13137.766} C_VEL
LIN {X 0,Y 360.533,Z 592.583,A -85,B 0,C 180,E1 -13138.883,E2 -13138.883} C_VEL
LIN {X 0,Y 360.495,Z 592.382,A -85,B 0,C 180,E1 -13140,E2 -13140} C_VEL
LIN {X 0,Y 360.497,Z 591.744,A -85,B 0,C 180,E1 -13141.117,E2 -13141.117} C_VEL
LIN {X 0,Y 360.516,Z 590.688,A -85,B 0,C 180,E1 -13142.235,E2 -13142.235} C_VEL
LIN {X 0,Y 360.527,Z 589.228,A -85,B 0,C 180,E1 -13143.353,E2 -13143.353} C_VEL
LIN {X 0,Y 360.712,Z 586.215,A -85,B 0,C 180,E1 -13145.03,E2 -13145.03} C_VEL
LIN {X 0,Y 360.922,Z 581.366,A -85,B 0,C 180,E1 -13146.99,E2 -13146.99} C_VEL
LIN {X 0,Y 361.247,Z 576.005,A -85,B 0,C 180,E1 -13148.672,E2 -13148.672} C_VEL
LIN {X 0,Y 361.818,Z 569.283,A -85,B 0,C 180,E1 -13150.351,E2 -13150.351} C_VEL
LIN {X 0,Y 362.488,Z 561.01,A -85,B 0,C 180,E1 -13152.03,E2 -13152.03} C_VEL
LIN {X 0,Y 363.488,Z 550.839,A -85,B 0,C 180,E1 -13153.701,E2 -13153.701} C_VEL
LIN {X 0,Y 364.483,Z 540.124,A -85,B 0,C 180,E1 -13155.118,E2 -13155.118} C_VEL
LIN {X 0,Y 365.311,Z 528.846,A -85,B 0,C 180,E1 -13156.342,E2 -13156.342} C_VEL
LIN {X 0,Y 366.188,Z 517.842,A -85,B 0,C 180,E1 -13157.306,E2 -13157.306} C_VEL
LIN {X 0,Y 366.533,Z 512.283,A -85,B 0,C 180,E1 -13157.722,E2 -13157.722} C_VEL
LIN {X 0,Y 364.216,Z 499.267,A -85,B 0,C 180,E1 -13158.645,E2 -13158.645} C_VEL
LIN {X 0,Y 361.501,Z 485.306,A -85,B 0,C 180,E1 -13159.421,E2 -13159.421} C_VEL
LIN {X 0,Y 361.041,Z 482.618,A -85,B 0,C 180,E1 -13159.574,E2 -13159.574} C_VEL
LIN {X 0,Y 361.214,Z 477.33,A -85,B 0,C 180,E1 -13162.901,E2 -13162.901} C_VEL
LIN {X 0,Y 361.532,Z 471.572,A -85,B 0,C 180,E1 -13166.59,E2 -13166.59} C_VEL
LIN {X 0,Y 361.748,Z 467.794,A -85,B 0,C 180,E1 -13169.058,E2 -13169.058} C_VEL
LIN {X 0,Y 361.953,Z 463.944,A -85,B 0,C 180,E1 -13171.618,E2 -13171.618} C_VEL
LIN {X 0,Y 362.124,Z 460.06,A -85,B 0,C 180,E1 -13174.251,E2 -13174.251} C_VEL
LIN {X 0,Y 362.112,Z 455.721,A -85,B 0,C 180,E1 -13177.273,E2 -13177.273} C_VEL
LIN {X 0,Y 361.999,Z 454.021,A -85,B 0,C 180,E1 -13178.565,E2 -13178.565} C_VEL
LIN {X 0,Y 361.843,Z 454.036,A -85,B 0,C 180,E1 -13182.828,E2 -13182.828} C_VEL
LIN {X 0,Y 361.91,Z 454.041,A -85,B 0,C 180,E1 -13187.006,E2 -13187.006} C_VEL
LIN {X 0,Y 362.999,Z 460.366,A -85,B 0,C 180,E1 -13190.288,E2 -13190.288} C_VEL
LIN {X 0,Y 363.213,Z 464.787,A -85,B 0,C 180,E1 -13192.498,E2 -13192.498} C_VEL
LIN {X 0,Y 362.906,Z 471.61,A -85,B 0,C 180,E1 -13195.831,E2 -13195.831} C_VEL
LIN {X 0,Y 362.499,Z 479.781,A -85,B 0,C 180,E1 -13199.728,E2 -13199.728} C_VEL
LIN {X 0,Y 362.159,Z 487.964,A -85,B 0,C 180,E1 -13203.49,E2 -13203.49} C_VEL
LIN {X 0,Y 361.952,Z 493.203,A -85,B 0,C 180,E1 -13205.735,E2 -13205.735} C_VEL
LIN {X 0,Y 366.27,Z 508.443,A -85,B 0,C 180,E1 -13206.483,E2 -13206.483} C_VEL
LIN {X 0,Y 369.195,Z 522.077,A -85,B 0,C 180,E1 -13207.307,E2 -13207.307} C_VEL
LIN {X 0,Y 370.705,Z 531.808,A -85,B 0,C 180,E1 -13208.001,E2 -13208.001} C_VEL
LIN {X 0,Y 369.614,Z 545.246,A -85,B 0,C 180,E1 -13208.966,E2 -13208.966} C_VEL
LIN {X 0,Y 368.308,Z 557.282,A -85,B 0,C 180,E1 -13210.056,E2 -13210.056} C_VEL
LIN {X 0,Y 366.726,Z 569.484,A -85,B 0,C 180,E1 -13211.42,E2 -13211.42} C_VEL
LIN {X 0,Y 365.358,Z 580.383,A -85,B 0,C 180,E1 -13212.94,E2 -13212.94} C_VEL
LIN {X 0,Y 363.981,Z 590.284,A -85,B 0,C 180,E1 -13214.622,E2 -13214.622} C_VEL
LIN {X 0,Y 363.091,Z 598.322,A -85,B 0,C 180,E1 -13216.283,E2 -13216.283} C_VEL
LIN {X 0,Y 361.955,Z 606.1,A -85,B 0,C 180,E1 -13218.235,E2 -13218.235} C_VEL
LIN {X 0,Y 361.346,Z 611.552,A -85,B 0,C 180,E1 -13219.917,E2 -13219.917} C_VEL
LIN {X 0,Y 360.773,Z 617.256,A -85,B 0,C 180,E1 -13222.161,E2 -13222.161} C_VEL
LIN {X 0,Y 360.612,Z 620.275,A -85,B 0,C 180,E1 -13223.693,E2 -13223.693} C_VEL
LIN {X 0,Y 360.389,Z 622.936,A -85,B 0,C 180,E1 -13225.525,E2 -13225.525} C_VEL
LIN {X 0,Y 360.257,Z 624.973,A -85,B 0,C 180,E1 -13227.763,E2 -13227.763} C_VEL
LIN {X 0,Y 360.274,Z 625.675,A -85,B 0,C 180,E1 -13229.999,E2 -13229.999} C_VEL
LIN {X 0,Y 360.256,Z 625.045,A -85,B 0,C 180,E1 -13232.235,E2 -13232.235} C_VEL
LIN {X 0,Y 360.387,Z 623.07,A -85,B 0,C 180,E1 -13234.472,E2 -13234.472} C_VEL
LIN {X 0,Y 360.609,Z 619.709,A -85,B 0,C 180,E1 -13236.714,E2 -13236.714} C_VEL
LIN {X 0,Y 361.018,Z 614.862,A -85,B 0,C 180,E1 -13238.958,E2 -13238.958} C_VEL
LIN {X 0,Y 361.673,Z 608.386,A -85,B 0,C 180,E1 -13241.203,E2 -13241.203} C_VEL
LIN {X 0,Y 362.696,Z 601.166,A -85,B 0,C 180,E1 -13243.159,E2 -13243.159} C_VEL
LIN {X 0,Y 363.722,Z 592.317,A -85,B 0,C 180,E1 -13245.09,E2 -13245.09} C_VEL
LIN {X 0,Y 365.03,Z 582.761,A -85,B 0,C 180,E1 -13246.784,E2 -13246.784} C_VEL
LIN {X 0,Y 366.392,Z 572.338,A -85,B 0,C 180,E1 -13248.305,E2 -13248.305} C_VEL
LIN {X 0,Y 367.906,Z 560.834,A -85,B 0,C 180,E1 -13249.673,E2 -13249.673} C_VEL
LIN {X 0,Y 369.328,Z 548.076,A -85,B 0,C 180,E1 -13250.902,E2 -13250.902} C_VEL
LIN {X 0,Y 370.502,Z 535.091,A -85,B 0,C 180,E1 -13251.89,E2 -13251.89} C_VEL
LIN {X 0,Y 370.561,Z 530.327,A -85,B 0,C 180,E1 -13252.209,E2 -13252.209} C_VEL
LIN {X 0,Y 368.13,Z 516.589,A -85,B 0,C 180,E1 -13253.146,E2 -13253.146} C_VEL
LIN {X 0,Y 366.115,Z 507.88,A -85,B 0,C 180,E1 -13253.65,E2 -13253.65} C_VEL
LIN {X 0,Y 364.259,Z 502.905,A -85,B 0,C 180,E1 -13253.991,E2 -13253.991} C_VEL
LIN {X 0,Y 361.645,Z 498.646,A -85,B 0,C 180,E1 -13254.451,E2 -13254.451} C_VEL
LIN {X 0,Y 358.051,Z 493.954,A -85,B 0,C 180,E1 -13255.235,E2 -13255.235} C_VEL
LIN {X 0,Y 355.982,Z 491.091,A -85,B 0,C 180,E1 -13255.956,E2 -13255.956} C_VEL
LIN {X 0,Y 355.253,Z 489.508,A -85,B 0,C 180,E1 -13256.496,E2 -13256.496} C_VEL
LIN {X 0,Y 355.172,Z 488.834,A -85,B 0,C 180,E1 -13256.78,E2 -13256.78} C_VEL
LIN {X 0,Y 355.512,Z 481.298,A -85,B 0,C 180,E1 -13260.27,E2 -13260.27} C_VEL
LIN {X 0,Y 355.954,Z 472.76,A -85,B 0,C 180,E1 -13264.375,E2 -13264.375} C_VEL
LIN {X 0,Y 356.262,Z 465.697,A -85,B 0,C 180,E1 -13267.9,E2 -13267.9} C_VEL
LIN {X 0,Y 356.209,Z 462.129,A -85,B 0,C 180,E1 -13269.693,E2 -13269.693} C_VEL
LIN {X 0,Y 354.894,Z 454.904,A -85,B 0,C 180,E1 -13273.503,E2 -13273.503} C_VEL
LIN {X 0,Y 354.835,Z 454.914,A -85,B 0,C 180,E1 -13277.122,E2 -13277.122} C_VEL
LIN {X 0,Y 354.83,Z 454.91,A -85,B 0,C 180,E1 -13280.668,E2 -13280.668} C_VEL
LIN {X 0,Y 354.814,Z 454.914,A -85,B 0,C 180,E1 -13284.299,E2 -13284.299} C_VEL
LIN {X 0,Y 354.79,Z 454.918,A -85,B 0,C 180,E1 -13287.667,E2 -13287.667} C_VEL
LIN {X 0,Y 354.86,Z 454.909,A -85,B 0,C 180,E1 -13290.62,E2 -13290.62} C_VEL
LIN {X 0,Y 354.89,Z 454.9,A -85,B 0,C 180,E1 -13294.172,E2 -13294.172} C_VEL
LIN {X 0,Y 354.841,Z 454.897,A -85,B 0,C 180,E1 -13297.894,E2 -13297.894} C_VEL
LIN {X 0,Y 354.913,Z 454.9,A -85,B 0,C 180,E1 -13301.89,E2 -13301.89} C_VEL
LIN {X 0,Y 354.933,Z 454.899,A -85,B 0,C 180,E1 -13305.98,E2 -13305.98} C_VEL
LIN {X 0,Y 354.972,Z 454.893,A -85,B 0,C 180,E1 -13309.736,E2 -13309.736} C_VEL
LIN {X 0,Y 355.104,Z 454.873,A -85,B 0,C 180,E1 -13312.037,E2 -13312.037} C_VEL
LIN {X 0,Y 355.088,Z 454.876,A -85,B 0,C 180,E1 -13314.321,E2 -13314.321} C_VEL
LIN {X 0,Y 355.237,Z 454.858,A -85,B 0,C 180,E1 -13317.732,E2 -13317.732} C_VEL
LIN {X 0,Y 355.388,Z 454.841,A -85,B 0,C 180,E1 -13320,E2 -13320} C_VEL
LIN {X 0,Y 355.236,Z 454.851,A -85,B 0,C 180,E1 -13322.268,E2 -13322.268} C_VEL
LIN {X 0,Y 355.127,Z 454.874,A -85,B 0,C 180,E1 -13326.819,E2 -13326.819} C_VEL
LIN {X 0,Y 355.006,Z 454.883,A -85,B 0,C 180,E1 -13329.113,E2 -13329.113} C_VEL
LIN {X 0,Y 354.916,Z 454.894,A -85,B 0,C 180,E1 -13332.581,E2 -13332.581} C_VEL
LIN {X 0,Y 354.879,Z 454.897,A -85,B 0,C 180,E1 -13336.096,E2 -13336.096} C_VEL
LIN {X 0,Y 354.891,Z 454.889,A -85,B 0,C 180,E1 -13338.473,E2 -13338.473} C_VEL
LIN {X 0,Y 354.825,Z 454.909,A -85,B 0,C 180,E1 -13342.107,E2 -13342.107} C_VEL
LIN {X 0,Y 354.889,Z 454.904,A -85,B 0,C 180,E1 -13345.828,E2 -13345.828} C_VEL
LIN {X 0,Y 354.845,Z 454.909,A -85,B 0,C 180,E1 -13349.679,E2 -13349.679} C_VEL
LIN {X 0,Y 354.797,Z 454.915,A -85,B 0,C 180,E1 -13353.703,E2 -13353.703} C_VEL
LIN {X 0,Y 354.793,Z 454.913,A -85,B 0,C 180,E1 -13356.46,E2 -13356.46} C_VEL
LIN {X 0,Y 354.815,Z 454.913,A -85,B 0,C 180,E1 -13359.425,E2 -13359.425} C_VEL
LIN {X 0,Y 354.826,Z 454.914,A -85,B 0,C 180,E1 -13362.876,E2 -13362.876} C_VEL
LIN {X 0,Y 354.801,Z 454.916,A -85,B 0,C 180,E1 -13366.111,E2 -13366.111} C_VEL
LIN {X 0,Y 354.859,Z 455.043,A -85,B 0,C 180,E1 -13367.342,E2 -13367.342} C_VEL
LIN {X 0,Y 356.196,Z 461.888,A -85,B 0,C 180,E1 -13370.85,E2 -13370.85} C_VEL
LIN {X 0,Y 357.6,Z 469.522,A -85,B 0,C 180,E1 -13374.568,E2 -13374.568} C_VEL
LIN {X 0,Y 358.15,Z 472.826,A -85,B 0,C 180,E1 -13376.121,E2 -13376.121} C_VEL
LIN {X 0,Y 357.808,Z 477.028,A -85,B 0,C 180,E1 -13377.974,E2 -13377.974} C_VEL
LIN {X 0,Y 356.6,Z 485.884,A -85,B 0,C 180,E1 -13381.773,E2 -13381.773} C_VEL
LIN {X 0,Y 355.651,Z 494.479,A -85,B 0,C 180,E1 -13385.38,E2 -13385.38} C_VEL
LIN {X 0,Y 359.727,Z 512.224,A -85,B 0,C 180,E1 -13386.145,E2 -13386.145} C_VEL
LIN {X 0,Y 362.254,Z 526.329,A -85,B 0,C 180,E1 -13386.94,E2 -13386.94} C_VEL
LIN {X 0,Y 363.52,Z 537.596,A -85,B 0,C 180,E1 -13387.704,E2 -13387.704} C_VEL
LIN {X 0,Y 362.365,Z 550.385,A -85,B 0,C 180,E1 -13388.616,E2 -13388.616} C_VEL
LIN {X 0,Y 360.968,Z 563.234,A -85,B 0,C 180,E1 -13389.784,E2 -13389.784} C_VEL
LIN {X 0,Y 359.382,Z 575.439,A -85,B 0,C 180,E1 -13391.177,E2 -13391.177} C_VEL
LIN {X 0,Y 358.039,Z 585.482,A -85,B 0,C 180,E1 -13392.583,E2 -13392.583} C_VEL
LIN {X 0,Y 356.686,Z 595.447,A -85,B 0,C 180,E1 -13394.282,E2 -13394.282} C_VEL
LIN {X 0,Y 355.655,Z 603.49,A -85,B 0,C 180,E1 -13395.942,E2 -13395.942} C_VEL
LIN {X 0,Y 354.88,Z 610.573,A -85,B 0,C 180,E1 -13397.71,E2 -13397.71} C_VEL
LIN {X 0,Y 354.098,Z 617.086,A -85,B 0,C 180,E1 -13399.712,E2 -13399.712} C_VEL
LIN {X 0,Y 353.554,Z 622.847,A -85,B 0,C 180,E1 -13402.003,E2 -13402.003} C_VEL
LIN {X 0,Y 353.328,Z 627.029,A -85,B 0,C 180,E1 -13404.294,E2 -13404.294} C_VEL
LIN {X 0,Y 353.224,Z 629.757,A -85,B 0,C 180,E1 -13406.579,E2 -13406.579} C_VEL
LIN {X 0,Y 353.211,Z 631.108,A -85,B 0,C 180,E1 -13408.861,E2 -13408.861} C_VEL
LIN {X 0,Y 353.213,Z 631.103,A -85,B 0,C 180,E1 -13411.142,E2 -13411.142} C_VEL
LIN {X 0,Y 353.225,Z 629.741,A -85,B 0,C 180,E1 -13413.423,E2 -13413.423} C_VEL
LIN {X 0,Y 353.33,Z 627.005,A -85,B 0,C 180,E1 -13415.709,E2 -13415.709} C_VEL
LIN {X 0,Y 353.557,Z 622.818,A -85,B 0,C 180,E1 -13418,E2 -13418} C_VEL
LIN {X 0,Y 354.097,Z 617.05,A -85,B 0,C 180,E1 -13420.291,E2 -13420.291} C_VEL
LIN {X 0,Y 354.866,Z 610.525,A -85,B 0,C 180,E1 -13422.294,E2 -13422.294} C_VEL
LIN {X 0,Y 355.665,Z 603.4,A -85,B 0,C 180,E1 -13424.068,E2 -13424.068} C_VEL
LIN {X 0,Y 356.7,Z 595.375,A -85,B 0,C 180,E1 -13425.72,E2 -13425.72} C_VEL
LIN {X 0,Y 358.084,Z 585.395,A -85,B 0,C 180,E1 -13427.417,E2 -13427.417} C_VEL
LIN {X 0,Y 360.666,Z 568.798,A -85,B 0,C 180,E1 -13429.791,E2 -13429.791} C_VEL
LIN {X 0,Y 362.677,Z 555.992,A -85,B 0,C 180,E1 -13431.286,E2 -13431.286} C_VEL
LIN {X 0,Y 364.644,Z 542.923,A -85,B 0,C 180,E1 -13432.525,E2 -13432.525} C_VEL
LIN {X 0,Y 365.194,Z 536.904,A -85,B 0,C 180,E1 -13433.039,E2 -13433.039} C_VEL
LIN {X 0,Y 364.503,Z 525.233,A -85,B 0,C 180,E1 -13434.075,E2 -13434.075} C_VEL
LIN {X 0,Y 362.433,Z 514.048,A -85,B 0,C 180,E1 -13435.089,E2 -13435.089} C_VEL
LIN {X 0,Y 359.043,Z 502.263,A -85,B 0,C 180,E1 -13436.198,E2 -13436.198} C_VEL
LIN {X 0,Y 357.17,Z 496.5,A -85,B 0,C 180,E1 -13436.745,E2 -13436.745} C_VEL
LIN {X 0,Y 357.555,Z 494.195,A -85,B 0,C 180,E1 -13437.809,E2 -13437.809} C_VEL
LIN {X 0,Y 359.109,Z 487.947,A -85,B 0,C 180,E1 -13441.241,E2 -13441.241} C_VEL
LIN {X 0,Y 359.942,Z 484.866,A -85,B 0,C 180,E1 -13443.143,E2 -13443.143} C_VEL
LIN {X 0,Y 360.228,Z 482.318,A -85,B 0,C 180,E1 -13444.974,E2 -13444.974} C_VEL
LIN {X 0,Y 359.91,Z 479.769,A -85,B 0,C 180,E1 -13447.255,E2 -13447.255} C_VEL
LIN {X 0,Y 359.505,Z 477.123,A -85,B 0,C 180,E1 -13450.322,E2 -13450.322} C_VEL
LIN {X 0,Y 359.069,Z 475.331,A -85,B 0,C 180,E1 -13453.598,E2 -13453.598} C_VEL
LIN {X 0,Y 358.829,Z 474.561,A -85,B 0,C 180,E1 -13456.725,E2 -13456.725} C_VEL
LIN {X 0,Y 358.733,Z 474.65,A -85,B 0,C 180,E1 -13459.825,E2 -13459.825} C_VEL
LIN {X 0,Y 358.561,Z 475.453,A -85,B 0,C 180,E1 -13462.583,E2 -13462.583} C_VEL
LIN {X 0,Y 358.402,Z 476.097,A -85,B 0,C 180,E1 -13463.965,E2 -13463.965} C_VEL
LIN {X 0,Y 357.703,Z 477.815,A -85,B 0,C 180,E1 -13466.624,E2 -13466.624} C_VEL
LIN {X 0,Y 356.847,Z 480.648,A -85,B 0,C 180,E1 -13470.064,E2 -13470.064} C_VEL
LIN {X 0,Y 356.2,Z 483.527,A -85,B 0,C 180,E1 -13473.012,E2 -13473.012} C_VEL
LIN {X 0,Y 355.727,Z 486.755,A -85,B 0,C 180,E1 -13475.798,E2 -13475.798} C_VEL
LIN {X 0,Y 357.016,Z 490.111,A -85,B 0,C 180,E1 -13476.195,E2 -13476.195} C_VEL
LIN {X 0,Y 361.746,Z 502.253,A -85,B 0,C 180,E1 -13477.693,E2 -13477.693} C_VEL
LIN {X 0,Y 364.401,Z 512.409,A -85,B 0,C 180,E1 -13478.873,E2 -13478.873} C_VEL
LIN {X 0,Y 365.714,Z 520.205,A -85,B 0,C 180,E1 -13479.763,E2 -13479.763} C_VEL
LIN {X 0,Y 363.874,Z 532.706,A -85,B 0,C 180,E1 -13480.978,E2 -13480.978} C_VEL
LIN {X 0,Y 361.791,Z 545.592,A -85,B 0,C 180,E1 -13482.549,E2 -13482.549} C_VEL
LIN {X 0,Y 359.938,Z 556.07,A -85,B 0,C 180,E1 -13484.136,E2 -13484.136} C_VEL
LIN {X 0,Y 358.488,Z 563.678,A -85,B 0,C 180,E1 -13485.525,E2 -13485.525} C_VEL
LIN {X 0,Y 356.974,Z 572.476,A -85,B 0,C 180,E1 -13487.493,E2 -13487.493} C_VEL
LIN {X 0,Y 355.934,Z 578.53,A -85,B 0,C 180,E1 -13489.189,E2 -13489.189} C_VEL
LIN {X 0,Y 355.127,Z 583.392,A -85,B 0,C 180,E1 -13490.891,E2 -13490.891} C_VEL
LIN {X 0,Y 354.277,Z 588.226,A -85,B 0,C 180,E1 -13493.164,E2 -13493.164} C_VEL
LIN {X 0,Y 353.888,Z 590.031,A -85,B 0,C 180,E1 -13494.301,E2 -13494.301} C_VEL
LIN {X 0,Y 353.805,Z 591.37,A -85,B 0,C 180,E1 -13495.443,E2 -13495.443} C_VEL
LIN {X 0,Y 353.735,Z 592.29,A -85,B 0,C 180,E1 -13496.583,E2 -13496.583} C_VEL
LIN {X 0,Y 353.595,Z 592.829,A -85,B 0,C 180,E1 -13497.722,E2 -13497.722} C_VEL
LIN {X 0,Y 353.473,Z 592.977,A -85,B 0,C 180,E1 -13498.861,E2 -13498.861} C_VEL
LIN {X 0,Y 353.432,Z 592.713,A -85,B 0,C 180,E1 -13500,E2 -13500} C_VEL
LIN {X 0,Y 353.403,Z 592.012,A -85,B 0,C 180,E1 -13501.14,E2 -13501.14} C_VEL
LIN {X 0,Y 353.42,Z 590.909,A -85,B 0,C 180,E1 -13502.279,E2 -13502.279} C_VEL
LIN {X 0,Y 353.442,Z 589.402,A -85,B 0,C 180,E1 -13503.42,E2 -13503.42} C_VEL
LIN {X 0,Y 353.633,Z 586.296,A -85,B 0,C 180,E1 -13505.131,E2 -13505.131} C_VEL
LIN {X 0,Y 353.851,Z 581.694,A -85,B 0,C 180,E1 -13507.002,E2 -13507.002} C_VEL
LIN {X 0,Y 354.218,Z 575.843,A -85,B 0,C 180,E1 -13508.845,E2 -13508.845} C_VEL
LIN {X 0,Y 354.806,Z 568.998,A -85,B 0,C 180,E1 -13510.558,E2 -13510.558} C_VEL
LIN {X 0,Y 355.493,Z 560.595,A -85,B 0,C 180,E1 -13512.27,E2 -13512.27} C_VEL
LIN {X 0,Y 356.347,Z 552.135,A -85,B 0,C 180,E1 -13513.69,E2 -13513.69} C_VEL
LIN {X 0,Y 357.268,Z 542.717,A -85,B 0,C 180,E1 -13515.01,E2 -13515.01} C_VEL
LIN {X 0,Y 358.226,Z 530.726,A -85,B 0,C 180,E1 -13516.381,E2 -13516.381} C_VEL
LIN {X 0,Y 359.227,Z 518.476,A -85,B 0,C 180,E1 -13517.506,E2 -13517.506} C_VEL
LIN {X 0,Y 359.371,Z 511.942,A -85,B 0,C 180,E1 -13518.013,E2 -13518.013} C_VEL
LIN {X 0,Y 356.819,Z 497.888,A -85,B 0,C 180,E1 -13519.014,E2 -13519.014} C_VEL
LIN {X 0,Y 354.186,Z 484.242,A -85,B 0,C 180,E1 -13519.757,E2 -13519.757} C_VEL
LIN {X 0,Y 353.965,Z 482.812,A -85,B 0,C 180,E1 -13519.84,E2 -13519.84} C_VEL
LIN {X 0,Y 354.189,Z 477.276,A -85,B 0,C 180,E1 -13523.382,E2 -13523.382} C_VEL
LIN {X 0,Y 354.488,Z 471.532,A -85,B 0,C 180,E1 -13527.129,E2 -13527.129} C_VEL
LIN {X 0,Y 354.709,Z 467.686,A -85,B 0,C 180,E1 -13529.692,E2 -13529.692} C_VEL
LIN {X 0,Y 354.961,Z 463.8,A -85,B 0,C 180,E1 -13532.316,E2 -13532.316} C_VEL
LIN {X 0,Y 355.108,Z 458.845,A -85,B 0,C 180,E1 -13535.762,E2 -13535.762} C_VEL
LIN {X 0,Y 354.973,Z 454.895,A -85,B 0,C 180,E1 -13538.675,E2 -13538.675} C_VEL
LIN {X 0,Y 354.794,Z 454.914,A -85,B 0,C 180,E1 -13542.867,E2 -13542.867} C_VEL
LIN {X 0,Y 354.876,Z 455.056,A -85,B 0,C 180,E1 -13546.699,E2 -13546.699} C_VEL
LIN {X 0,Y 355.783,Z 459.981,A -85,B 0,C 180,E1 -13549.316,E2 -13549.316} C_VEL
LIN {X 0,Y 356.284,Z 464.284,A -85,B 0,C 180,E1 -13551.545,E2 -13551.545} C_VEL
LIN {X 0,Y 355.971,Z 471.386,A -85,B 0,C 180,E1 -13555.07,E2 -13555.07} C_VEL
LIN {X 0,Y 355.64,Z 477.806,A -85,B 0,C 180,E1 -13558.185,E2 -13558.185} C_VEL
LIN {X 0,Y 355.311,Z 485.155,A -85,B 0,C 180,E1 -13561.658,E2 -13561.658} C_VEL
LIN {X 0,Y 354.96,Z 492.995,A -85,B 0,C 180,E1 -13565.196,E2 -13565.196} C_VEL
LIN {X 0,Y 359.759,Z 510.016,A -85,B 0,C 180,E1 -13566.091,E2 -13566.091} C_VEL
LIN {X 0,Y 362.655,Z 523.894,A -85,B 0,C 180,E1 -13566.979,E2 -13566.979} C_VEL
LIN {X 0,Y 364.068,Z 533.069,A -85,B 0,C 180,E1 -13567.662,E2 -13567.662} C_VEL
LIN {X 0,Y 362.976,Z 545.288,A -85,B 0,C 180,E1 -13568.563,E2 -13568.563} C_VEL
LIN {X 0,Y 361.634,Z 557.328,A -85,B 0,C 180,E1 -13569.671,E2 -13569.671} C_VEL
LIN {X 0,Y 359.971,Z 569.534,A -85,B 0,C 180,E1 -13571.058,E2 -13571.058} C_VEL
LIN {X 0,Y 358.551,Z 580.435,A -85,B 0,C 180,E1 -13572.606,E2 -13572.606} C_VEL
LIN {X 0,Y 357.118,Z 590.24,A -85,B 0,C 180,E1 -13574.299,E2 -13574.299} C_VEL
LIN {X 0,Y 356.275,Z 597.153,A -85,B 0,C 180,E1 -13575.723,E2 -13575.723} C_VEL
LIN {X 0,Y 355.119,Z 605.163,A -85,B 0,C 180,E1 -13577.715,E2 -13577.715} C_VEL
LIN {X 0,Y 354.322,Z 611.608,A -85,B 0,C 180,E1 -13579.715,E2 -13579.715} C_VEL
LIN {X 0,Y 353.72,Z 617.312,A -85,B 0,C 180,E1 -13582.004,E2 -13582.004} C_VEL
LIN {X 0,Y 353.404,Z 621.46,A -85,B 0,C 180,E1 -13584.292,E2 -13584.292} C_VEL
LIN {X 0,Y 353.222,Z 624.179,A -85,B 0,C 180,E1 -13586.577,E2 -13586.577} C_VEL
LIN {X 0,Y 353.155,Z 625.546,A -85,B 0,C 180,E1 -13588.858,E2 -13588.858} C_VEL
LIN {X 0,Y 353.155,Z 625.583,A -85,B 0,C 180,E1 -13591.139,E2 -13591.139} C_VEL
LIN {X 0,Y 353.221,Z 624.282,A -85,B 0,C 180,E1 -13593.421,E2 -13593.421} C_VEL
LIN {X 0,Y 353.4,Z 621.623,A -85,B 0,C 180,E1 -13595.705,E2 -13595.705} C_VEL
LIN {X 0,Y 353.704,Z 617.533,A -85,B 0,C 180,E1 -13597.994,E2 -13597.994} C_VEL
LIN {X 0,Y 354.286,Z 611.891,A -85,B 0,C 180,E1 -13600.283,E2 -13600.283} C_VEL
LIN {X 0,Y 355.097,Z 605.519,A -85,B 0,C 180,E1 -13602.283,E2 -13602.283} C_VEL
LIN {X 0,Y 356.063,Z 598.81,A -85,B 0,C 180,E1 -13603.991,E2 -13603.991} C_VEL
LIN {X 0,Y 357.023,Z 590.905,A -85,B 0,C 180,E1 -13605.673,E2 -13605.673} C_VEL
LIN {X 0,Y 358.484,Z 581.058,A -85,B 0,C 180,E1 -13607.394,E2 -13607.394} C_VEL
LIN {X 0,Y 359.902,Z 570.285,A -85,B 0,C 180,E1 -13608.942,E2 -13608.942} C_VEL
LIN {X 0,Y 361.566,Z 558.314,A -85,B 0,C 180,E1 -13610.33,E2 -13610.33} C_VEL
LIN {X 0,Y 362.871,Z 546.547,A -85,B 0,C 180,E1 -13611.437,E2 -13611.437} C_VEL
LIN {X 0,Y 364.031,Z 533.505,A -85,B 0,C 180,E1 -13612.412,E2 -13612.412} C_VEL
LIN {X 0,Y 362.629,Z 523.73,A -85,B 0,C 180,E1 -13613.135,E2 -13613.135} C_VEL
LIN {X 0,Y 359.684,Z 509.636,A -85,B 0,C 180,E1 -13614.033,E2 -13614.033} C_VEL
LIN {X 0,Y 355.43,Z 495.096,A -85,B 0,C 180,E1 -13614.8,E2 -13614.8} C_VEL
LIN {X 0,Y 354.954,Z 492.995,A -85,B 0,C 180,E1 -13614.911,E2 -13614.911} C_VEL
LIN {X 0,Y 355.172,Z 488.834,A -85,B 0,C 180,E1 -13616.78,E2 -13616.78} C_VEL
LIN {X 0,Y 354.602,Z 486.981,A -85,B 0,C 180,E1 -13617.68,E2 -13617.68} C_VEL
LIN {X 0,Y 351.894,Z 484.274,A -85,B 0,C 180,E1 -13619.165,E2 -13619.165} C_VEL
LIN {X 0,Y 349.595,Z 482.178,A -85,B 0,C 180,E1 -13620.369,E2 -13620.369} C_VEL
LIN {X 0,Y 348.651,Z 480.438,A -85,B 0,C 180,E1 -13621.292,E2 -13621.292} C_VEL
LIN {X 0,Y 348.599,Z 479.812,A -85,B 0,C 180,E1 -13621.602,E2 -13621.602} C_VEL
LIN {X 0,Y 349.008,Z 472.834,A -85,B 0,C 180,E1 -13625.02,E2 -13625.02} C_VEL
LIN {X 0,Y 349.358,Z 465.779,A -85,B 0,C 180,E1 -13628.579,E2 -13628.579} C_VEL
LIN {X 0,Y 349.138,Z 462.844,A -85,B 0,C 180,E1 -13630.099,E2 -13630.099} C_VEL
LIN {X 0,Y 347.851,Z 455.782,A -85,B 0,C 180,E1 -13633.919,E2 -13633.919} C_VEL
LIN {X 0,Y 347.811,Z 455.788,A -85,B 0,C 180,E1 -13636.669,E2 -13636.669} C_VEL
LIN {X 0,Y 347.778,Z 455.787,A -85,B 0,C 180,E1 -13640.164,E2 -13640.164} C_VEL
LIN {X 0,Y 347.781,Z 455.79,A -85,B 0,C 180,E1 -13644.124,E2 -13644.124} C_VEL
LIN {X 0,Y 347.756,Z 455.788,A -85,B 0,C 180,E1 -13648.301,E2 -13648.301} C_VEL
LIN {X 0,Y 347.798,Z 455.788,A -85,B 0,C 180,E1 -13650.989,E2 -13650.989} C_VEL
LIN {X 0,Y 347.822,Z 455.775,A -85,B 0,C 180,E1 -13653.607,E2 -13653.607} C_VEL
LIN {X 0,Y 347.788,Z 455.787,A -85,B 0,C 180,E1 -13656.162,E2 -13656.162} C_VEL
LIN {X 0,Y 347.826,Z 455.781,A -85,B 0,C 180,E1 -13659.91,E2 -13659.91} C_VEL
LIN {X 0,Y 347.857,Z 455.778,A -85,B 0,C 180,E1 -13662.359,E2 -13662.359} C_VEL
LIN {X 0,Y 347.887,Z 455.777,A -85,B 0,C 180,E1 -13665.97,E2 -13665.97} C_VEL
LIN {X 0,Y 347.923,Z 455.772,A -85,B 0,C 180,E1 -13669.525,E2 -13669.525} C_VEL
LIN {X 0,Y 348.064,Z 455.749,A -85,B 0,C 180,E1 -13671.874,E2 -13671.874} C_VEL
LIN {X 0,Y 348.063,Z 455.752,A -85,B 0,C 180,E1 -13674.206,E2 -13674.206} C_VEL
LIN {X 0,Y 348.199,Z 455.735,A -85,B 0,C 180,E1 -13677.686,E2 -13677.686} C_VEL
LIN {X 0,Y 348.358,Z 455.717,A -85,B 0,C 180,E1 -13680,E2 -13680} C_VEL
LIN {X 0,Y 348.198,Z 455.726,A -85,B 0,C 180,E1 -13682.313,E2 -13682.313} C_VEL
LIN {X 0,Y 348.095,Z 455.75,A -85,B 0,C 180,E1 -13686.958,E2 -13686.958} C_VEL
LIN {X 0,Y 347.958,Z 455.756,A -85,B 0,C 180,E1 -13689.299,E2 -13689.299} C_VEL
LIN {X 0,Y 347.884,Z 455.771,A -85,B 0,C 180,E1 -13692.84,E2 -13692.84} C_VEL
LIN {X 0,Y 347.829,Z 455.769,A -85,B 0,C 180,E1 -13696.432,E2 -13696.432} C_VEL
LIN {X 0,Y 347.841,Z 455.772,A -85,B 0,C 180,E1 -13698.861,E2 -13698.861} C_VEL
LIN {X 0,Y 347.764,Z 455.789,A -85,B 0,C 180,E1 -13702.58,E2 -13702.58} C_VEL
LIN {X 0,Y 347.802,Z 455.785,A -85,B 0,C 180,E1 -13705.109,E2 -13705.109} C_VEL
LIN {X 0,Y 347.802,Z 455.784,A -85,B 0,C 180,E1 -13707.695,E2 -13707.695} C_VEL
LIN {X 0,Y 347.755,Z 455.794,A -85,B 0,C 180,E1 -13710.347,E2 -13710.347} C_VEL
LIN {X 0,Y 347.735,Z 455.796,A -85,B 0,C 180,E1 -13714.465,E2 -13714.465} C_VEL
LIN {X 0,Y 347.77,Z 455.791,A -85,B 0,C 180,E1 -13717.991,E2 -13717.991} C_VEL
LIN {X 0,Y 347.775,Z 455.789,A -85,B 0,C 180,E1 -13721.827,E2 -13721.827} C_VEL
LIN {X 0,Y 347.79,Z 455.788,A -85,B 0,C 180,E1 -13725.013,E2 -13725.013} C_VEL
LIN {X 0,Y 347.802,Z 455.872,A -85,B 0,C 180,E1 -13726.984,E2 -13726.984} C_VEL
LIN {X 0,Y 349.173,Z 462.953,A -85,B 0,C 180,E1 -13730.694,E2 -13730.694} C_VEL
LIN {X 0,Y 350.571,Z 470.517,A -85,B 0,C 180,E1 -13734.455,E2 -13734.455} C_VEL
LIN {X 0,Y 351.098,Z 473.553,A -85,B 0,C 180,E1 -13735.913,E2 -13735.913} C_VEL
LIN {X 0,Y 350.773,Z 478.007,A -85,B 0,C 180,E1 -13737.933,E2 -13737.933} C_VEL
LIN {X 0,Y 349.534,Z 486.774,A -85,B 0,C 180,E1 -13741.768,E2 -13741.768} C_VEL
LIN {X 0,Y 348.744,Z 493.917,A -85,B 0,C 180,E1 -13744.84,E2 -13744.84} C_VEL
LIN {X 0,Y 352.927,Z 512.01,A -85,B 0,C 180,E1 -13745.648,E2 -13745.648} C_VEL
LIN {X 0,Y 355.522,Z 526.467,A -85,B 0,C 180,E1 -13746.485,E2 -13746.485} C_VEL
LIN {X 0,Y 356.862,Z 538.848,A -85,B 0,C 180,E1 -13747.352,E2 -13747.352} C_VEL
LIN {X 0,Y 355.618,Z 551.721,A -85,B 0,C 180,E1 -13748.309,E2 -13748.309} C_VEL
LIN {X 0,Y 354.145,Z 564.529,A -85,B 0,C 180,E1 -13749.529,E2 -13749.529} C_VEL
LIN {X 0,Y 352.505,Z 576.462,A -85,B 0,C 180,E1 -13750.947,E2 -13750.947} C_VEL
LIN {X 0,Y 350.993,Z 587.213,A -85,B 0,C 180,E1 -13752.523,E2 -13752.523} C_VEL
LIN {X 0,Y 349.611,Z 596.88,A -85,B 0,C 180,E1 -13754.255,E2 -13754.255} C_VEL
LIN {X 0,Y 348.535,Z 604.881,A -85,B 0,C 180,E1 -13755.999,E2 -13755.999} C_VEL
LIN {X 0,Y 347.766,Z 611.527,A -85,B 0,C 180,E1 -13757.751,E2 -13757.751} C_VEL
LIN {X 0,Y 347.068,Z 617.032,A -85,B 0,C 180,E1 -13759.501,E2 -13759.501} C_VEL
LIN {X 0,Y 346.499,Z 622.793,A -85,B 0,C 180,E1 -13761.839,E2 -13761.839} C_VEL
LIN {X 0,Y 346.248,Z 626.975,A -85,B 0,C 180,E1 -13764.177,E2 -13764.177} C_VEL
LIN {X 0,Y 346.148,Z 629.702,A -85,B 0,C 180,E1 -13766.509,E2 -13766.509} C_VEL
LIN {X 0,Y 346.111,Z 631.052,A -85,B 0,C 180,E1 -13768.838,E2 -13768.838} C_VEL
LIN {X 0,Y 346.113,Z 631.047,A -85,B 0,C 180,E1 -13771.165,E2 -13771.165} C_VEL
LIN {X 0,Y 346.149,Z 629.685,A -85,B 0,C 180,E1 -13773.494,E2 -13773.494} C_VEL
LIN {X 0,Y 346.249,Z 626.949,A -85,B 0,C 180,E1 -13775.826,E2 -13775.826} C_VEL
LIN {X 0,Y 346.502,Z 622.763,A -85,B 0,C 180,E1 -13778.164,E2 -13778.164} C_VEL
LIN {X 0,Y 347.065,Z 616.994,A -85,B 0,C 180,E1 -13780.502,E2 -13780.502} C_VEL
LIN {X 0,Y 347.884,Z 610.47,A -85,B 0,C 180,E1 -13782.544,E2 -13782.544} C_VEL
LIN {X 0,Y 348.864,Z 602.373,A -85,B 0,C 180,E1 -13784.58,E2 -13784.58} C_VEL
LIN {X 0,Y 350.07,Z 593.818,A -85,B 0,C 180,E1 -13786.325,E2 -13786.325} C_VEL
LIN {X 0,Y 352.776,Z 576.575,A -85,B 0,C 180,E1 -13789.192,E2 -13789.192} C_VEL
LIN {X 0,Y 354.974,Z 564.308,A -85,B 0,C 180,E1 -13790.879,E2 -13790.879} C_VEL
LIN {X 0,Y 357.155,Z 551.682,A -85,B 0,C 180,E1 -13792.291,E2 -13792.291} C_VEL
LIN {X 0,Y 358.964,Z 538.504,A -85,B 0,C 180,E1 -13793.507,E2 -13793.507} C_VEL
LIN {X 0,Y 358.416,Z 526.861,A -85,B 0,C 180,E1 -13794.607,E2 -13794.607} C_VEL
LIN {X 0,Y 356.224,Z 514.726,A -85,B 0,C 180,E1 -13795.79,E2 -13795.79} C_VEL
LIN {X 0,Y 353.086,Z 503.685,A -85,B 0,C 180,E1 -13796.92,E2 -13796.92} C_VEL
LIN {X 0,Y 350.643,Z 496.507,A -85,B 0,C 180,E1 -13797.678,E2 -13797.678} C_VEL
LIN {X 0,Y 350.546,Z 495.982,A -85,B 0,C 180,E1 -13797.732,E2 -13797.732} C_VEL
LIN {X 0,Y 352.184,Z 489.711,A -85,B 0,C 180,E1 -13801.256,E2 -13801.256} C_VEL
LIN {X 0,Y 353.087,Z 486.528,A -85,B 0,C 180,E1 -13803.281,E2 -13803.281} C_VEL
LIN {X 0,Y 353.323,Z 483.786,A -85,B 0,C 180,E1 -13805.36,E2 -13805.36} C_VEL
LIN {X 0,Y 352.955,Z 480.932,A -85,B 0,C 180,E1 -13808.118,E2 -13808.118} C_VEL
LIN {X 0,Y 352.563,Z 478.627,A -85,B 0,C 180,E1 -13811.135,E2 -13811.135} C_VEL
LIN {X 0,Y 352.197,Z 477.134,A -85,B 0,C 180,E1 -13814.301,E2 -13814.301} C_VEL
LIN {X 0,Y 351.979,Z 476.521,A -85,B 0,C 180,E1 -13817.629,E2 -13817.629} C_VEL
LIN {X 0,Y 351.891,Z 476.906,A -85,B 0,C 180,E1 -13821.163,E2 -13821.163} C_VEL
LIN {X 0,Y 351.665,Z 477.609,A -85,B 0,C 180,E1 -13823.163,E2 -13823.163} C_VEL
LIN {X 0,Y 351.027,Z 479.142,A -85,B 0,C 180,E1 -13825.903,E2 -13825.903} C_VEL
LIN {X 0,Y 349.991,Z 482.176,A -85,B 0,C 180,E1 -13829.867,E2 -13829.867} C_VEL
LIN {X 0,Y 349.103,Z 485.843,A -85,B 0,C 180,E1 -13833.711,E2 -13833.711} C_VEL
LIN {X 0,Y 348.914,Z 487.051,A -85,B 0,C 180,E1 -13834.762,E2 -13834.762} C_VEL
LIN {X 0,Y 350.193,Z 490.33,A -85,B 0,C 180,E1 -13835.195,E2 -13835.195} C_VEL
LIN {X 0,Y 350.813,Z 491.439,A -85,B 0,C 180,E1 -13835.371,E2 -13835.371} C_VEL
LIN {X 0,Y 355.267,Z 502.963,A -85,B 0,C 180,E1 -13836.912,E2 -13836.912} C_VEL
LIN {X 0,Y 357.917,Z 512.369,A -85,B 0,C 180,E1 -13838.094,E2 -13838.094} C_VEL
LIN {X 0,Y 359.493,Z 521.734,A -85,B 0,C 180,E1 -13839.241,E2 -13839.241} C_VEL
LIN {X 0,Y 357.632,Z 533.944,A -85,B 0,C 180,E1 -13840.484,E2 -13840.484} C_VEL
LIN {X 0,Y 355.7,Z 544.969,A -85,B 0,C 180,E1 -13841.854,E2 -13841.854} C_VEL
LIN {X 0,Y 353.945,Z 554.352,A -85,B 0,C 180,E1 -13843.267,E2 -13843.267} C_VEL
LIN {X 0,Y 351.967,Z 563.722,A -85,B 0,C 180,E1 -13844.955,E2 -13844.955} C_VEL
LIN {X 0,Y 350.392,Z 572.515,A -85,B 0,C 180,E1 -13846.959,E2 -13846.959} C_VEL
LIN {X 0,Y 349.028,Z 579.482,A -85,B 0,C 180,E1 -13848.972,E2 -13848.972} C_VEL
LIN {X 0,Y 348.183,Z 584.233,A -85,B 0,C 180,E1 -13850.707,E2 -13850.707} C_VEL
LIN {X 0,Y 347.56,Z 587.563,A -85,B 0,C 180,E1 -13852.241,E2 -13852.241} C_VEL
LIN {X 0,Y 346.856,Z 590.661,A -85,B 0,C 180,E1 -13854.185,E2 -13854.185} C_VEL
LIN {X 0,Y 346.671,Z 592.784,A -85,B 0,C 180,E1 -13856.513,E2 -13856.513} C_VEL
LIN {X 0,Y 346.523,Z 593.275,A -85,B 0,C 180,E1 -13857.675,E2 -13857.675} C_VEL
LIN {X 0,Y 346.395,Z 593.369,A -85,B 0,C 180,E1 -13858.838,E2 -13858.838} C_VEL
LIN {X 0,Y 346.351,Z 593.018,A -85,B 0,C 180,E1 -13860,E2 -13860} C_VEL
LIN {X 0,Y 346.308,Z 592.266,A -85,B 0,C 180,E1 -13861.163,E2 -13861.163} C_VEL
LIN {X 0,Y 346.324,Z 591.115,A -85,B 0,C 180,E1 -13862.326,E2 -13862.326} C_VEL
LIN {X 0,Y 346.414,Z 588.584,A -85,B 0,C 180,E1 -13864.072,E2 -13864.072} C_VEL
LIN {X 0,Y 346.612,Z 584.269,A -85,B 0,C 180,E1 -13866.162,E2 -13866.162} C_VEL
LIN {X 0,Y 346.948,Z 578.641,A -85,B 0,C 180,E1 -13868.152,E2 -13868.152} C_VEL
LIN {X 0,Y 347.578,Z 571.2,A -85,B 0,C 180,E1 -13870.191,E2 -13870.191} C_VEL
LIN {X 0,Y 348.245,Z 563.224,A -85,B 0,C 180,E1 -13871.938,E2 -13871.938} C_VEL
LIN {X 0,Y 349.232,Z 553.38,A -85,B 0,C 180,E1 -13873.678,E2 -13873.678} C_VEL
LIN {X 0,Y 350.215,Z 543.417,A -85,B 0,C 180,E1 -13875.122,E2 -13875.122} C_VEL
LIN {X 0,Y 351.117,Z 532.478,A -85,B 0,C 180,E1 -13876.423,E2 -13876.423} C_VEL
LIN {X 0,Y 352.08,Z 520.539,A -85,B 0,C 180,E1 -13877.573,E2 -13877.573} C_VEL
LIN {X 0,Y 352.516,Z 513.456,A -85,B 0,C 180,E1 -13878.15,E2 -13878.15} C_VEL
LIN {X 0,Y 350.155,Z 500.283,A -85,B 0,C 180,E1 -13879.137,E2 -13879.137} C_VEL
LIN {X 0,Y 347.447,Z 485.94,A -85,B 0,C 180,E1 -13879.977,E2 -13879.977} C_VEL
LIN {X 0,Y 346.912,Z 482.975,A -85,B 0,C 180,E1 -13880.145,E2 -13880.145} C_VEL
LIN {X 0,Y 347.19,Z 477.211,A -85,B 0,C 180,E1 -13883.882,E2 -13883.882} C_VEL
LIN {X 0,Y 347.462,Z 471.427,A -85,B 0,C 180,E1 -13887.724,E2 -13887.724} C_VEL
LIN {X 0,Y 347.692,Z 467.55,A -85,B 0,C 180,E1 -13890.354,E2 -13890.354} C_VEL
LIN {X 0,Y 347.962,Z 463.637,A -85,B 0,C 180,E1 -13893.048,E2 -13893.048} C_VEL
LIN {X 0,Y 348.065,Z 459.288,A -85,B 0,C 180,E1 -13896.13,E2 -13896.13} C_VEL
LIN {X 0,Y 347.936,Z 455.772,A -85,B 0,C 180,E1 -13898.768,E2 -13898.768} C_VEL
LIN {X 0,Y 347.757,Z 455.794,A -85,B 0,C 180,E1 -13901.83,E2 -13901.83} C_VEL
LIN {X 0,Y 347.794,Z 455.797,A -85,B 0,C 180,E1 -13906.238,E2 -13906.238} C_VEL
LIN {X 0,Y 348.768,Z 461.079,A -85,B 0,C 180,E1 -13909.086,E2 -13909.086} C_VEL
LIN {X 0,Y 349.33,Z 465.528,A -85,B 0,C 180,E1 -13911.414,E2 -13911.414} C_VEL
LIN {X 0,Y 349.002,Z 472.578,A -85,B 0,C 180,E1 -13914.975,E2 -13914.975} C_VEL
LIN {X 0,Y 348.609,Z 479.536,A -85,B 0,C 180,E1 -13918.387,E2 -13918.387} C_VEL
LIN {X 0,Y 348.306,Z 486.486,A -85,B 0,C 180,E1 -13921.693,E2 -13921.693} C_VEL
LIN {X 0,Y 348.01,Z 493.186,A -85,B 0,C 180,E1 -13924.698,E2 -13924.698} C_VEL
LIN {X 0,Y 352.395,Z 508.357,A -85,B 0,C 180,E1 -13925.494,E2 -13925.494} C_VEL
LIN {X 0,Y 355.417,Z 521.681,A -85,B 0,C 180,E1 -13926.351,E2 -13926.351} C_VEL
LIN {X 0,Y 357.419,Z 534.194,A -85,B 0,C 180,E1 -13927.3,E2 -13927.3} C_VEL
LIN {X 0,Y 356.3,Z 546.107,A -85,B 0,C 180,E1 -13928.21,E2 -13928.21} C_VEL
LIN {X 0,Y 354.789,Z 558.753,A -85,B 0,C 180,E1 -13929.413,E2 -13929.413} C_VEL
LIN {X 0,Y 353.09,Z 570.641,A -85,B 0,C 180,E1 -13930.826,E2 -13930.826} C_VEL
LIN {X 0,Y 351.753,Z 580.487,A -85,B 0,C 180,E1 -13932.259,E2 -13932.259} C_VEL
LIN {X 0,Y 350.251,Z 590.294,A -85,B 0,C 180,E1 -13933.983,E2 -13933.983} C_VEL
LIN {X 0,Y 349.324,Z 597.381,A -85,B 0,C 180,E1 -13935.474,E2 -13935.474} C_VEL
LIN {X 0,Y 348.176,Z 605.218,A -85,B 0,C 180,E1 -13937.466,E2 -13937.466} C_VEL
LIN {X 0,Y 347.313,Z 611.663,A -85,B 0,C 180,E1 -13939.505,E2 -13939.505} C_VEL
LIN {X 0,Y 346.664,Z 617.368,A -85,B 0,C 180,E1 -13941.84,E2 -13941.84} C_VEL
LIN {X 0,Y 346.339,Z 621.516,A -85,B 0,C 180,E1 -13944.175,E2 -13944.175} C_VEL
LIN {X 0,Y 346.148,Z 624.235,A -85,B 0,C 180,E1 -13946.506,E2 -13946.506} C_VEL
LIN {X 0,Y 346.058,Z 625.602,A -85,B 0,C 180,E1 -13948.835,E2 -13948.835} C_VEL
LIN {X 0,Y 346.058,Z 625.638,A -85,B 0,C 180,E1 -13951.162,E2 -13951.162} C_VEL
LIN {X 0,Y 346.146,Z 624.337,A -85,B 0,C 180,E1 -13953.491,E2 -13953.491} C_VEL
LIN {X 0,Y 346.337,Z 621.677,A -85,B 0,C 180,E1 -13955.822,E2 -13955.822} C_VEL
LIN {X 0,Y 346.651,Z 617.587,A -85,B 0,C 180,E1 -13958.157,E2 -13958.157} C_VEL
LIN {X 0,Y 347.275,Z 611.944,A -85,B 0,C 180,E1 -13960.493,E2 -13960.493} C_VEL
LIN {X 0,Y 348.15,Z 605.57,A -85,B 0,C 180,E1 -13962.532,E2 -13962.532} C_VEL
LIN {X 0,Y 349.106,Z 598.916,A -85,B 0,C 180,E1 -13964.262,E2 -13964.262} C_VEL
LIN {X 0,Y 350.406,Z 589.347,A -85,B 0,C 180,E1 -13966.306,E2 -13966.306} C_VEL
LIN {X 0,Y 351.965,Z 579.323,A -85,B 0,C 180,E1 -13968.028,E2 -13968.028} C_VEL
LIN {X 0,Y 353.509,Z 568.102,A -85,B 0,C 180,E1 -13969.6,E2 -13969.6} C_VEL
LIN {X 0,Y 355.203,Z 555.659,A -85,B 0,C 180,E1 -13971.004,E2 -13971.004} C_VEL
LIN {X 0,Y 356.611,Z 543.113,A -85,B 0,C 180,E1 -13972.14,E2 -13972.14} C_VEL
LIN {X 0,Y 357.421,Z 533.956,A -85,B 0,C 180,E1 -13972.819,E2 -13972.819} C_VEL
LIN {X 0,Y 355.228,Z 520.664,A -85,B 0,C 180,E1 -13973.82,E2 -13973.82} C_VEL
LIN {X 0,Y 352.089,Z 507.147,A -85,B 0,C 180,E1 -13974.678,E2 -13974.678} C_VEL
LIN {X 0,Y 347.996,Z 493.023,A -85,B 0,C 180,E1 -13975.434,E2 -13975.434} C_VEL
LIN {X 0,Y 348.4,Z 485.33,A -85,B 0,C 180,E1 -13978.954,E2 -13978.954} C_VEL
LIN {X 0,Y 348.599,Z 479.812,A -85,B 0,C 180,E1 -13981.602,E2 -13981.602} C_VEL
LIN {X 0,Y 348.031,Z 478.043,A -85,B 0,C 180,E1 -13982.525,E2 -13982.525} C_VEL
LIN {X 0,Y 345.36,Z 475.495,A -85,B 0,C 180,E1 -13984.047,E2 -13984.047} C_VEL
LIN {X 0,Y 343.11,Z 473.501,A -85,B 0,C 180,E1 -13985.281,E2 -13985.281} C_VEL
LIN {X 0,Y 342.207,Z 471.822,A -85,B 0,C 180,E1 -13986.226,E2 -13986.226} C_VEL
LIN {X 0,Y 342.169,Z 471.209,A -85,B 0,C 180,E1 -13986.542,E2 -13986.542} C_VEL
LIN {X 0,Y 342.411,Z 466.942,A -85,B 0,C 180,E1 -13988.744,E2 -13988.744} C_VEL
LIN {X 0,Y 341.873,Z 462.489,A -85,B 0,C 180,E1 -13991.132,E2 -13991.132} C_VEL
LIN {X 0,Y 340.805,Z 456.66,A -85,B 0,C 180,E1 -13994.323,E2 -13994.323} C_VEL
LIN {X 0,Y 340.745,Z 456.667,A -85,B 0,C 180,E1 -13997.943,E2 -13997.943} C_VEL
LIN {X 0,Y 340.727,Z 456.666,A -85,B 0,C 180,E1 -14000.251,E2 -14000.251} C_VEL
LIN {X 0,Y 340.703,Z 456.672,A -85,B 0,C 180,E1 -14003.558,E2 -14003.558} C_VEL
LIN {X 0,Y 340.687,Z 456.669,A -85,B 0,C 180,E1 -14006.153,E2 -14006.153} C_VEL
LIN {X 0,Y 340.767,Z 456.664,A -85,B 0,C 180,E1 -14010.332,E2 -14010.332} C_VEL
LIN {X 0,Y 340.796,Z 456.65,A -85,B 0,C 180,E1 -14013.019,E2 -14013.019} C_VEL
LIN {X 0,Y 340.77,Z 456.663,A -85,B 0,C 180,E1 -14015.639,E2 -14015.639} C_VEL
LIN {X 0,Y 340.767,Z 456.659,A -85,B 0,C 180,E1 -14019.475,E2 -14019.475} C_VEL
LIN {X 0,Y 340.849,Z 456.651,A -85,B 0,C 180,E1 -14021.984,E2 -14021.984} C_VEL
LIN {X 0,Y 340.859,Z 456.65,A -85,B 0,C 180,E1 -14025.704,E2 -14025.704} C_VEL
LIN {X 0,Y 340.865,Z 456.652,A -85,B 0,C 180,E1 -14029.306,E2 -14029.306} C_VEL
LIN {X 0,Y 341.068,Z 456.626,A -85,B 0,C 180,E1 -14032.898,E2 -14032.898} C_VEL
LIN {X 0,Y 341.161,Z 456.612,A -85,B 0,C 180,E1 -14037.639,E2 -14037.639} C_VEL
LIN {X 0,Y 341.307,Z 456.595,A -85,B 0,C 180,E1 -14040,E2 -14040} C_VEL
LIN {X 0,Y 341.16,Z 456.601,A -85,B 0,C 180,E1 -14042.361,E2 -14042.361} C_VEL
LIN {X 0,Y 341.065,Z 456.625,A -85,B 0,C 180,E1 -14047.102,E2 -14047.102} C_VEL
LIN {X 0,Y 340.865,Z 456.626,A -85,B 0,C 180,E1 -14050.694,E2 -14050.694} C_VEL
LIN {X 0,Y 340.852,Z 456.652,A -85,B 0,C 180,E1 -14054.325,E2 -14054.325} C_VEL
LIN {X 0,Y 340.826,Z 456.64,A -85,B 0,C 180,E1 -14058.467,E2 -14058.467} C_VEL
LIN {X 0,Y 340.743,Z 456.664,A -85,B 0,C 180,E1 -14061.858,E2 -14061.858} C_VEL
LIN {X 0,Y 340.763,Z 456.662,A -85,B 0,C 180,E1 -14065.665,E2 -14065.665} C_VEL
LIN {X 0,Y 340.733,Z 456.664,A -85,B 0,C 180,E1 -14068.32,E2 -14068.32} C_VEL
LIN {X 0,Y 340.695,Z 456.67,A -85,B 0,C 180,E1 -14071.045,E2 -14071.045} C_VEL
LIN {X 0,Y 340.71,Z 456.671,A -85,B 0,C 180,E1 -14075.28,E2 -14075.28} C_VEL
LIN {X 0,Y 340.711,Z 456.669,A -85,B 0,C 180,E1 -14078.389,E2 -14078.389} C_VEL
LIN {X 0,Y 340.717,Z 456.667,A -85,B 0,C 180,E1 -14081.305,E2 -14081.305} C_VEL
LIN {X 0,Y 340.714,Z 456.671,A -85,B 0,C 180,E1 -14084.534,E2 -14084.534} C_VEL
LIN {X 0,Y 340.763,Z 456.831,A -85,B 0,C 180,E1 -14086.686,E2 -14086.686} C_VEL
LIN {X 0,Y 342.118,Z 463.837,A -85,B 0,C 180,E1 -14090.447,E2 -14090.447} C_VEL
LIN {X 0,Y 343.526,Z 471.387,A -85,B 0,C 180,E1 -14094.288,E2 -14094.288} C_VEL
LIN {X 0,Y 344.074,Z 474.53,A -85,B 0,C 180,E1 -14095.828,E2 -14095.828} C_VEL
LIN {X 0,Y 343.874,Z 477.884,A -85,B 0,C 180,E1 -14097.388,E2 -14097.388} C_VEL
LIN {X 0,Y 342.654,Z 486.329,A -85,B 0,C 180,E1 -14101.186,E2 -14101.186} C_VEL
LIN {X 0,Y 341.789,Z 493.328,A -85,B 0,C 180,E1 -14104.272,E2 -14104.272} C_VEL
LIN {X 0,Y 346.176,Z 512.244,A -85,B 0,C 180,E1 -14105.148,E2 -14105.148} C_VEL
LIN {X 0,Y 348.724,Z 526.189,A -85,B 0,C 180,E1 -14105.983,E2 -14105.983} C_VEL
LIN {X 0,Y 350.199,Z 539.096,A -85,B 0,C 180,E1 -14106.915,E2 -14106.915} C_VEL
LIN {X 0,Y 349.108,Z 551.046,A -85,B 0,C 180,E1 -14107.826,E2 -14107.826} C_VEL
LIN {X 0,Y 347.674,Z 563.16,A -85,B 0,C 180,E1 -14108.975,E2 -14108.975} C_VEL
LIN {X 0,Y 346.123,Z 574.262,A -85,B 0,C 180,E1 -14110.273,E2 -14110.273} C_VEL
LIN {X 0,Y 344.466,Z 585.39,A -85,B 0,C 180,E1 -14111.874,E2 -14111.874} C_VEL
LIN {X 0,Y 342.973,Z 595.349,A -85,B 0,C 180,E1 -14113.637,E2 -14113.637} C_VEL
LIN {X 0,Y 341.827,Z 603.04,A -85,B 0,C 180,E1 -14115.275,E2 -14115.275} C_VEL
LIN {X 0,Y 340.921,Z 610.469,A -85,B 0,C 180,E1 -14117.198,E2 -14117.198} C_VEL
LIN {X 0,Y 340.047,Z 616.979,A -85,B 0,C 180,E1 -14119.282,E2 -14119.282} C_VEL
LIN {X 0,Y 339.436,Z 622.739,A -85,B 0,C 180,E1 -14121.668,E2 -14121.668} C_VEL
LIN {X 0,Y 339.168,Z 626.92,A -85,B 0,C 180,E1 -14124.055,E2 -14124.055} C_VEL
LIN {X 0,Y 339.073,Z 629.646,A -85,B 0,C 180,E1 -14126.437,E2 -14126.437} C_VEL
LIN {X 0,Y 339.013,Z 630.997,A -85,B 0,C 180,E1 -14128.814,E2 -14128.814} C_VEL
LIN {X 0,Y 339.015,Z 630.991,A -85,B 0,C 180,E1 -14131.189,E2 -14131.189} C_VEL
LIN {X 0,Y 339.073,Z 629.629,A -85,B 0,C 180,E1 -14133.566,E2 -14133.566} C_VEL
LIN {X 0,Y 339.17,Z 626.893,A -85,B 0,C 180,E1 -14135.948,E2 -14135.948} C_VEL
LIN {X 0,Y 339.44,Z 622.707,A -85,B 0,C 180,E1 -14138.335,E2 -14138.335} C_VEL
LIN {X 0,Y 340.021,Z 616.938,A -85,B 0,C 180,E1 -14140.722,E2 -14140.722} C_VEL
LIN {X 0,Y 340.908,Z 610.415,A -85,B 0,C 180,E1 -14142.805,E2 -14142.805} C_VEL
LIN {X 0,Y 341.88,Z 602.844,A -85,B 0,C 180,E1 -14144.758,E2 -14144.758} C_VEL
LIN {X 0,Y 343.223,Z 593.765,A -85,B 0,C 180,E1 -14146.66,E2 -14146.66} C_VEL
LIN {X 0,Y 345.833,Z 579.209,A -85,B 0,C 180,E1 -14149.284,E2 -14149.284} C_VEL
LIN {X 0,Y 347.838,Z 568.713,A -85,B 0,C 180,E1 -14150.863,E2 -14150.863} C_VEL
LIN {X 0,Y 350.195,Z 556.116,A -85,B 0,C 180,E1 -14152.416,E2 -14152.416} C_VEL
LIN {X 0,Y 352.619,Z 542.173,A -85,B 0,C 180,E1 -14153.805,E2 -14153.805} C_VEL
LIN {X 0,Y 352.714,Z 532.762,A -85,B 0,C 180,E1 -14154.737,E2 -14154.737} C_VEL
LIN {X 0,Y 351.428,Z 521.937,A -85,B 0,C 180,E1 -14155.851,E2 -14155.851} C_VEL
LIN {X 0,Y 348.894,Z 510.796,A -85,B 0,C 180,E1 -14157.05,E2 -14157.05} C_VEL
LIN {X 0,Y 345.331,Z 499.717,A -85,B 0,C 180,E1 -14158.321,E2 -14158.321} C_VEL
LIN {X 0,Y 344.101,Z 495.71,A -85,B 0,C 180,E1 -14158.783,E2 -14158.783} C_VEL
LIN {X 0,Y 345.604,Z 490.449,A -85,B 0,C 180,E1 -14161.92,E2 -14161.92} C_VEL
LIN {X 0,Y 346.288,Z 487.836,A -85,B 0,C 180,E1 -14163.685,E2 -14163.685} C_VEL
LIN {X 0,Y 346.386,Z 484.959,A -85,B 0,C 180,E1 -14166.045,E2 -14166.045} C_VEL
LIN {X 0,Y 346.029,Z 482.154,A -85,B 0,C 180,E1 -14169.024,E2 -14169.024} C_VEL
LIN {X 0,Y 345.642,Z 480.098,A -85,B 0,C 180,E1 -14172.145,E2 -14172.145} C_VEL
LIN {X 0,Y 345.321,Z 478.87,A -85,B 0,C 180,E1 -14175.426,E2 -14175.426} C_VEL
LIN {X 0,Y 345.118,Z 478.556,A -85,B 0,C 180,E1 -14178.893,E2 -14178.893} C_VEL
LIN {X 0,Y 345.069,Z 478.809,A -85,B 0,C 180,E1 -14180.848,E2 -14180.848} C_VEL
LIN {X 0,Y 344.686,Z 479.803,A -85,B 0,C 180,E1 -14183.751,E2 -14183.751} C_VEL
LIN {X 0,Y 343.864,Z 481.662,A -85,B 0,C 180,E1 -14186.928,E2 -14186.928} C_VEL
LIN {X 0,Y 342.9,Z 484.479,A -85,B 0,C 180,E1 -14190.535,E2 -14190.535} C_VEL
LIN {X 0,Y 342.213,Z 487.457,A -85,B 0,C 180,E1 -14193.628,E2 -14193.628} C_VEL
LIN {X 0,Y 343.508,Z 490.811,A -85,B 0,C 180,E1 -14194.123,E2 -14194.123} C_VEL
LIN {X 0,Y 344.594,Z 493.116,A -85,B 0,C 180,E1 -14194.493,E2 -14194.493} C_VEL
LIN {X 0,Y 348.365,Z 502.307,A -85,B 0,C 180,E1 -14195.87,E2 -14195.87} C_VEL
LIN {X 0,Y 351.579,Z 513.008,A -85,B 0,C 180,E1 -14197.338,E2 -14197.338} C_VEL
LIN {X 0,Y 353.26,Z 522.72,A -85,B 0,C 180,E1 -14198.6,E2 -14198.6} C_VEL
LIN {X 0,Y 353.396,Z 524.435,A -85,B 0,C 180,E1 -14198.817,E2 -14198.817} C_VEL
LIN {X 0,Y 351.227,Z 536.494,A -85,B 0,C 180,E1 -14200.113,E2 -14200.113} C_VEL
LIN {X 0,Y 349.151,Z 547.258,A -85,B 0,C 180,E1 -14201.529,E2 -14201.529} C_VEL
LIN {X 0,Y 346.992,Z 557.783,A -85,B 0,C 180,E1 -14203.225,E2 -14203.225} C_VEL
LIN {X 0,Y 345.064,Z 566.533,A -85,B 0,C 180,E1 -14204.949,E2 -14204.949} C_VEL
LIN {X 0,Y 343.315,Z 574.805,A -85,B 0,C 180,E1 -14206.987,E2 -14206.987} C_VEL
LIN {X 0,Y 342.137,Z 580.519,A -85,B 0,C 180,E1 -14208.747,E2 -14208.747} C_VEL
LIN {X 0,Y 341.245,Z 585.09,A -85,B 0,C 180,E1 -14210.517,E2 -14210.517} C_VEL
LIN {X 0,Y 340.53,Z 588.453,A -85,B 0,C 180,E1 -14212.163,E2 -14212.163} C_VEL
LIN {X 0,Y 339.828,Z 591.29,A -85,B 0,C 180,E1 -14214.065,E2 -14214.065} C_VEL
LIN {X 0,Y 339.609,Z 593.295,A -85,B 0,C 180,E1 -14216.441,E2 -14216.441} C_VEL
LIN {X 0,Y 339.454,Z 593.725,A -85,B 0,C 180,E1 -14217.627,E2 -14217.627} C_VEL
LIN {X 0,Y 339.32,Z 593.73,A -85,B 0,C 180,E1 -14218.813,E2 -14218.813} C_VEL
LIN {X 0,Y 339.258,Z 593.32,A -85,B 0,C 180,E1 -14220,E2 -14220} C_VEL
LIN {X 0,Y 339.213,Z 592.514,A -85,B 0,C 180,E1 -14221.187,E2 -14221.187} C_VEL
LIN {X 0,Y 339.228,Z 591.309,A -85,B 0,C 180,E1 -14222.375,E2 -14222.375} C_VEL
LIN {X 0,Y 339.347,Z 588.673,A -85,B 0,C 180,E1 -14224.157,E2 -14224.157} C_VEL
LIN {X 0,Y 339.507,Z 585.036,A -85,B 0,C 180,E1 -14225.941,E2 -14225.941} C_VEL
LIN {X 0,Y 339.786,Z 580.31,A -85,B 0,C 180,E1 -14227.727,E2 -14227.727} C_VEL
LIN {X 0,Y 340.353,Z 573.255,A -85,B 0,C 180,E1 -14229.809,E2 -14229.809} C_VEL
LIN {X 0,Y 341.008,Z 565.669,A -85,B 0,C 180,E1 -14231.592,E2 -14231.592} C_VEL
LIN {X 0,Y 341.914,Z 556.402,A -85,B 0,C 180,E1 -14233.37,E2 -14233.37} C_VEL
LIN {X 0,Y 342.993,Z 545.896,A -85,B 0,C 180,E1 -14234.992,E2 -14234.992} C_VEL
LIN {X 0,Y 344.012,Z 534.191,A -85,B 0,C 180,E1 -14236.468,E2 -14236.468} C_VEL
LIN {X 0,Y 344.986,Z 522.605,A -85,B 0,C 180,E1 -14237.64,E2 -14237.64} C_VEL
LIN {X 0,Y 345.585,Z 515.76,A -85,B 0,C 180,E1 -14238.221,E2 -14238.221} C_VEL
LIN {X 0,Y 343.703,Z 503.878,A -85,B 0,C 180,E1 -14239.176,E2 -14239.176} C_VEL
LIN {X 0,Y 341.055,Z 489.757,A -85,B 0,C 180,E1 -14240.083,E2 -14240.083} C_VEL
LIN {X 0,Y 339.854,Z 483.143,A -85,B 0,C 180,E1 -14240.424,E2 -14240.424} C_VEL
LIN {X 0,Y 340.153,Z 476.811,A -85,B 0,C 180,E1 -14244.617,E2 -14244.617} C_VEL
LIN {X 0,Y 340.415,Z 472.674,A -85,B 0,C 180,E1 -14247.406,E2 -14247.406} C_VEL
LIN {X 0,Y 340.709,Z 467.397,A -85,B 0,C 180,E1 -14251.044,E2 -14251.044} C_VEL
LIN {X 0,Y 340.994,Z 462.541,A -85,B 0,C 180,E1 -14254.469,E2 -14254.469} C_VEL
LIN {X 0,Y 340.986,Z 458.461,A -85,B 0,C 180,E1 -14257.447,E2 -14257.447} C_VEL
LIN {X 0,Y 340.873,Z 456.651,A -85,B 0,C 180,E1 -14258.854,E2 -14258.854} C_VEL
LIN {X 0,Y 340.682,Z 456.672,A -85,B 0,C 180,E1 -14262.904,E2 -14262.904} C_VEL
LIN {X 0,Y 340.774,Z 456.752,A -85,B 0,C 180,E1 -14265.858,E2 -14265.858} C_VEL
LIN {X 0,Y 341.975,Z 463.377,A -85,B 0,C 180,E1 -14269.499,E2 -14269.499} C_VEL
LIN {X 0,Y 342.358,Z 466.727,A -85,B 0,C 180,E1 -14271.267,E2 -14271.267} C_VEL
LIN {X 0,Y 342.052,Z 473.789,A -85,B 0,C 180,E1 -14274.878,E2 -14274.878} C_VEL
LIN {X 0,Y 341.622,Z 480.809,A -85,B 0,C 180,E1 -14278.357,E2 -14278.357} C_VEL
LIN {X 0,Y 341.387,Z 486.437,A -85,B 0,C 180,E1 -14281.066,E2 -14281.066} C_VEL
LIN {X 0,Y 341.046,Z 493.106,A -85,B 0,C 180,E1 -14284.143,E2 -14284.143} C_VEL
LIN {X 0,Y 345.433,Z 508.145,A -85,B 0,C 180,E1 -14284.959,E2 -14284.959} C_VEL
LIN {X 0,Y 348.391,Z 520.716,A -85,B 0,C 180,E1 -14285.79,E2 -14285.79} C_VEL
LIN {X 0,Y 350.635,Z 534.331,A -85,B 0,C 180,E1 -14286.843,E2 -14286.843} C_VEL
LIN {X 0,Y 350.483,Z 538.428,A -85,B 0,C 180,E1 -14287.157,E2 -14287.157} C_VEL
LIN {X 0,Y 349.165,Z 550.739,A -85,B 0,C 180,E1 -14288.193,E2 -14288.193} C_VEL
LIN {X 0,Y 347.644,Z 562.596,A -85,B 0,C 180,E1 -14289.435,E2 -14289.435} C_VEL
LIN {X 0,Y 346.098,Z 572.787,A -85,B 0,C 180,E1 -14290.731,E2 -14290.731} C_VEL
LIN {X 0,Y 344.4,Z 584.039,A -85,B 0,C 180,E1 -14292.481,E2 -14292.481} C_VEL
LIN {X 0,Y 342.925,Z 593.261,A -85,B 0,C 180,E1 -14294.242,E2 -14294.242} C_VEL
LIN {X 0,Y 341.784,Z 602.033,A -85,B 0,C 180,E1 -14296.32,E2 -14296.32} C_VEL
LIN {X 0,Y 340.735,Z 608.23,A -85,B 0,C 180,E1 -14298.095,E2 -14298.095} C_VEL
LIN {X 0,Y 340.093,Z 613.31,A -85,B 0,C 180,E1 -14299.882,E2 -14299.882} C_VEL
LIN {X 0,Y 339.505,Z 618.633,A -85,B 0,C 180,E1 -14302.266,E2 -14302.266} C_VEL
LIN {X 0,Y 339.26,Z 621.572,A -85,B 0,C 180,E1 -14304.053,E2 -14304.053} C_VEL
LIN {X 0,Y 339.075,Z 624.291,A -85,B 0,C 180,E1 -14306.434,E2 -14306.434} C_VEL
LIN {X 0,Y 338.964,Z 625.658,A -85,B 0,C 180,E1 -14308.81,E2 -14308.81} C_VEL
LIN {X 0,Y 338.964,Z 625.694,A -85,B 0,C 180,E1 -14311.187,E2 -14311.187} C_VEL
LIN {X 0,Y 339.074,Z 624.392,A -85,B 0,C 180,E1 -14313.563,E2 -14313.563} C_VEL
LIN {X 0,Y 339.258,Z 621.732,A -85,B 0,C 180,E1 -14315.944,E2 -14315.944} C_VEL
LIN {X 0,Y 339.597,Z 617.641,A -85,B 0,C 180,E1 -14318.328,E2 -14318.328} C_VEL
LIN {X 0,Y 340.271,Z 611.997,A -85,B 0,C 180,E1 -14320.711,E2 -14320.711} C_VEL
LIN {X 0,Y 341.204,Z 605.622,A -85,B 0,C 180,E1 -14322.791,E2 -14322.791} C_VEL
LIN {X 0,Y 342.233,Z 598.306,A -85,B 0,C 180,E1 -14324.72,E2 -14324.72} C_VEL
LIN {X 0,Y 343.559,Z 589.395,A -85,B 0,C 180,E1 -14326.64,E2 -14326.64} C_VEL
LIN {X 0,Y 345.185,Z 579.368,A -85,B 0,C 180,E1 -14328.394,E2 -14328.394} C_VEL
LIN {X 0,Y 346.822,Z 568.143,A -85,B 0,C 180,E1 -14329.994,E2 -14329.994} C_VEL
LIN {X 0,Y 348.571,Z 555.791,A -85,B 0,C 180,E1 -14331.413,E2 -14331.413} C_VEL
